//     PlcTask Inputs/GVL_Safety.SafetyInputs/bStageCollectRightDoorCh1 <-> Module 1 (FSOE)/FSoE Inputs/FSOE/FSIN Module 1.Input
//     PlcTask Inputs/GVL_Safety.SafetyInputs/bStageCollectRightDoorCh2 <-> Module 1 (FSOE)/FSoE Inputs/FSOE/FSIN Module 2.Input
//     PlcTask Inputs/GVL_Safety.SafetyInputs/bStageCollectRightDoorFdbk <-> Module 1 (FSOE)/FSoE Inputs/FSOE/FSIN Module 3.Input
//   TE1063/TE1063 Instance <-> Device 3 (EtherCAT)/Term 1 (EK1100)/Term 6 (EL1918)
//     PlcTask Inputs/GVL_IO.nEL1918T06State <-> InfoData/State
//     PlcTask Inputs/GVL_Safety.SafetyInputs/bD4AccessDoorIntlckOSSD1 <-> Module 1 (FSOE)/FSoE Inputs/FSOE/FSIN Module 3.Input
//     PlcTask Inputs/GVL_Safety.SafetyInputs/bD4AccessDoorIntlckOSSD2 <-> Module 1 (FSOE)/FSoE Inputs/FSOE/FSIN Module 4.Input
//     PlcTask Inputs/GVL_Safety.SafetyInputs/bD5AccessDoorIntlckOSSD1 <-> Module 1 (FSOE)/FSoE Inputs/FSOE/FSIN Module 5.Input
//     PlcTask Inputs/GVL_Safety.SafetyInputs/bD5AccessDoorIntlckOSSD2 <-> Module 1 (FSOE)/FSoE Inputs/FSOE/FSIN Module 6.Input
//     PlcTask Inputs/GVL_Safety.SafetyInputs/bD6AccessDoorIntlckOSSD1 <-> Module 1 (FSOE)/FSoE Inputs/FSOE/FSIN Module 7.Input
//     PlcTask Inputs/GVL_Safety.SafetyInputs/bD6AccessDoorIntlckOSSD2 <-> Module 1 (FSOE)/FSoE Inputs/FSOE/FSIN Module 8.Input
//     PlcTask Inputs/GVL_Safety.SafetyInputs/bFestoMS6DumpValveFdbk <-> Module 1 (FSOE)/FSoE Inputs/FSOE/FSIN Module 2.Input
//     PlcTask Inputs/GVL_Safety.SafetyInputs/bFestoMS6ValveFdbk <-> Module 1 (FSOE)/FSoE Inputs/FSOE/FSIN Module 1.Input
//   TE1063/TE1063 Instance <-> Device 3 (EtherCAT)/Term 1 (EK1100)/Term 7 (EL2904)
//     PlcTask Inputs/GVL_IO.nEL2904T07State <-> InfoData/State
//   TE1063/TE1063 Instance <-> Device 3 (EtherCAT)/Term 1 (EK1100)/Term 8 (EL2904)
//     PlcTask Inputs/GVL_IO.nEL2904T08State <-> InfoData/State
//   TE1063/TE1063 Instance <-> Device 3 (EtherCAT)/Term 1 (EK1100)/Term 9 (EL1809)
//     PlcTask Inputs/GVL_IO.gDigInputs/b24VPowerSupplyOK <-> Channel 3/Input
//     PlcTask Inputs/GVL_IO.gDigInputs/b48VPowerSupplyOK <-> Channel 5/Input
//     PlcTask Inputs/GVL_IO.gDigInputs/b24VPowerSupplyOKBck <-> Channel 4/Input
//     PlcTask Inputs/GVL_IO.gDigInputs/b48VPowerSupplyOKBck <-> Channel 12/Input
//     PlcTask Inputs/GVL_IO.gDigInputs/bCalibrationBoxPresent <-> Channel 13/Input
//     PlcTask Inputs/GVL_IO.gDigInputs/bSampleRecovery_Horizontal_Home <-> Channel 8/Input
//     PlcTask Inputs/GVL_IO.gDigInputs/bSampleRecovery_Vertical_Home <-> Channel 7/Input
//     PlcTask Inputs/GVL_IO.gDigInputs/bStageCollection_Home <-> Channel 6/Input
//     PlcTask Inputs/GVL_IO.gDigInputs/bStartButton <-> Channel 1/Input
//     PlcTask Inputs/GVL_IO.gDigInputs/bStopButton <-> Channel 2/Input
//     PlcTask Inputs/GVL_IO.gDigInputs/bThroatJigPresent <-> Channel 14/Input
//     PlcTask Inputs/GVL_IO.gDigInputs/bUPSReady <-> Channel 10/Input
//     PlcTask Inputs/GVL_IO.gDigInputs/bUPSReplaceBattery <-> Channel 11/Input
//     PlcTask Inputs/GVL_IO.gDigInputs/bWasteOverflowSensor <-> Channel 9/Input
//     PlcTask Inputs/GVL_IO.nEL1809T09State <-> InfoData/State
//   TE1063/TE1063 Instance <-> Device 3 (EtherCAT)/Term 22 (EK1100)
//     Task_Services Inputs/GVL_IO.nEK1100T22State <-> InfoData/State
//   TE1063/TE1063 Instance <-> Device 3 (EtherCAT)/Term 22 (EK1100)/Term 23 (EL7062)
//     PlcTask Inputs/GVL_Motion.aPumps[1].Linear.iHomeSensor <-> DRV Info data 3 Channel 1/Info data 3
//     PlcTask Inputs/GVL_Motion.aPumps[1].Linear.nState <-> InfoData/State
//     PlcTask Inputs/GVL_Motion.aPumps[1].Rotary.nState <-> InfoData/State
//   TE1063/TE1063 Instance <-> Device 3 (EtherCAT)/Term 22 (EK1100)/Term 24 (EL7062)
//     PlcTask Inputs/GVL_Motion.aPumps[2].Linear.iHomeSensor <-> DRV Info data 3 Channel 1/Info data 3
//     PlcTask Inputs/GVL_Motion.aPumps[2].Linear.nState <-> InfoData/State
//     PlcTask Inputs/GVL_Motion.aPumps[2].Rotary.nState <-> InfoData/State
//   TE1063/TE1063 Instance <-> Device 3 (EtherCAT)/Term 22 (EK1100)/Term 25 (EL7062)
//     PlcTask Inputs/GVL_Motion.aPumps[3].Linear.iHomeSensor <-> DRV Info data 3 Channel 1/Info data 3
//     PlcTask Inputs/GVL_Motion.aPumps[3].Linear.nState <-> InfoData/State
//     PlcTask Inputs/GVL_Motion.aPumps[3].Rotary.nState <-> InfoData/State
//   TE1063/TE1063 Instance <-> Device 3 (EtherCAT)/Term 22 (EK1100)/Term 26 (EL7062)
//     PlcTask Inputs/GVL_Motion.aPumps[4].Linear.iHomeSensor <-> DRV Info data 3 Channel 1/Info data 3
//     PlcTask Inputs/GVL_Motion.aPumps[4].Linear.nState <-> InfoData/State
//     PlcTask Inputs/GVL_Motion.aPumps[4].Rotary.nState <-> InfoData/State
//   TE1063/TE1063 Instance <-> Device 3 (EtherCAT)/Term 22 (EK1100)/Term 27 (EL7062)
//     PlcTask Inputs/GVL_Motion.aPumps[5].Linear.iHomeSensor <-> DRV Info data 3 Channel 1/Info data 3
//     PlcTask Inputs/GVL_Motion.aPumps[5].Linear.nState <-> InfoData/State
//     PlcTask Inputs/GVL_Motion.aPumps[5].Rotary.nState <-> InfoData/State
//   TE1063/TE1063 Instance <-> Device 3 (EtherCAT)/Term 22 (EK1100)/Term 28 (EL7062)
//     PlcTask Inputs/GVL_Motion.aPumps[6].Linear.iHomeSensor <-> DRV Info data 3 Channel 1/Info data 3
//     PlcTask Inputs/GVL_Motion.aPumps[6].Linear.nState <-> InfoData/State
//     PlcTask Inputs/GVL_Motion.aPumps[6].Rotary.nState <-> InfoData/State
//   TE1063/TE1063 Instance <-> Device 3 (EtherCAT)/Term 22 (EK1100)/Term 29 (EL7062)
//     PlcTask Inputs/GVL_Motion.aPumps[7].Linear.iHomeSensor <-> DRV Info data 3 Channel 1/Info data 3
//     PlcTask Inputs/GVL_Motion.aPumps[7].Linear.nState <-> InfoData/State
//     PlcTask Inputs/GVL_Motion.aPumps[7].Rotary.nState <-> InfoData/State
//   TE1063/TE1063 Instance <-> Device 3 (EtherCAT)/Term 22 (EK1100)/Term 30 (EL7062)
//     PlcTask Inputs/GVL_Motion.aPumps[8].Linear.iHomeSensor <-> DRV Info data 3 Channel 1/Info data 3
//     PlcTask Inputs/GVL_Motion.aPumps[8].Linear.nState <-> InfoData/State
//     PlcTask Inputs/GVL_Motion.aPumps[8].Rotary.nState <-> InfoData/State
//   TE1063/TE1063 Instance <-> Device 3 (EtherCAT)/Term 22 (EK1100)/Term 31 (EL7062)
//     PlcTask Inputs/GVL_Motion.aPumps[9].Linear.iHomeSensor <-> DRV Info data 3 Channel 1/Info data 3
//     PlcTask Inputs/GVL_Motion.aPumps[9].Linear.nState <-> InfoData/State
//     PlcTask Inputs/GVL_Motion.aPumps[9].Rotary.nState <-> InfoData/State
//   TE1063/TE1063 Instance <-> Device 3 (EtherCAT)/Term 22 (EK1100)/Term 32 (EL7062)
//     PlcTask Inputs/GVL_Motion.aPumps[10].Linear.iHomeSensor <-> DRV Info data 3 Channel 1/Info data 3
//     PlcTask Inputs/GVL_Motion.aPumps[10].Linear.nState <-> InfoData/State
//     PlcTask Inputs/GVL_Motion.aPumps[10].Rotary.nState <-> InfoData/State
//   TE1063/TE1063 Instance <-> Device 3 (EtherCAT)/Term 33 (AX8620-0000-0105)
//     Task_Services Inputs/GVL_IO.nAX8620T33State <-> InfoData/State
//   TE1063/TE1063 Instance <-> Device 3 (EtherCAT)/Term 33 (AX8620-0000-0105)/Drive 34 (AX8108-0100-0106)
//     PlcTask Inputs/GVL_Motion.M1Motor.nState <-> InfoData/State
//     PlcTask Outputs/GVL_Motion.M1Motor.bTS_ErrorAck <-> Device (Safety)/Standard Outputdata/ChA_Connection_Input.ERR_ACK FSoE Connection_3
//     PlcTask Outputs/GVL_Motion.M1Motor.bTS_Run <-> Device (Safety)/Standard Outputdata/ChA_Connection_Input.RUN FSoE Connection_2
//   TE1063/TE1063 Instance <-> Device 5 (EL6631)/dl-pn1
//     PlcTask Inputs/GVL_IO.gProfinetInput/bCurrentValueInvalid <-> API/Term 3 (GT2-***)/Subterm 5 (GT2-***)/Inputs/Sensor Status/Current_Value_Invalid
//     PlcTask Inputs/GVL_IO.gProfinetInput/bCurrentValueOverRange <-> API/Term 3 (GT2-***)/Subterm 5 (GT2-***)/Inputs/Sensor Status/Current_Value_Over_Range
//     PlcTask Inputs/GVL_IO.gProfinetInput/bCurrentValueUnerRange <-> API/Term 3 (GT2-***)/Subterm 5 (GT2-***)/Inputs/Sensor Status/Current_Value_Under_Range
//     PlcTask Inputs/GVL_IO.gProfinetInput/bErrorStatus <-> API/Term 3 (GT2-***)/Subterm 5 (GT2-***)/Inputs/Sensor Status/Error_Status
//     PlcTask Inputs/GVL_IO.gProfinetInput/bWarningStatus <-> API/Term 3 (GT2-***)/Subterm 5 (GT2-***)/Inputs/Sensor Status/Warning_Status
//     PlcTask Inputs/GVL_IO.gProfinetInput/iCurrentValue <-> API/Term 3 (GT2-***)/Subterm 5 (GT2-***)/Inputs/Current Value
//     PlcTask Inputs/GVL_IO.gProfinetInput/iPnIoBoxState <-> Inputs/PnIoBoxState
//   TE1063/TE1063 Instance <-> Device 6 (EtherCAT)/Box 10 (AMI8000-0100)
//     PlcTask Inputs/GVL_Motion.aValves[3].nState <-> InfoData/State
//     PlcTask Outputs/GVL_Safety.iM6STOErrorAck <-> Module 1 (SAFETY)/SAFETY Standard Outputdata/Standard In Var 3
//     PlcTask Outputs/GVL_Safety.iM6STORun <-> Module 1 (SAFETY)/SAFETY Standard Outputdata/Standard In Var 2
//   TE1063/TE1063 Instance <-> Device 6 (EtherCAT)/Box 11 (AMI8000-0100)
//     PlcTask Inputs/GVL_Motion.aValves[4].nState <-> InfoData/State
//     PlcTask Outputs/GVL_Safety.iM7STOErrorAck <-> Module 1 (SAFETY)/SAFETY Standard Outputdata/Standard In Var 3
//     PlcTask Outputs/GVL_Safety.iM7STORun <-> Module 1 (SAFETY)/SAFETY Standard Outputdata/Standard In Var 2
//   TE1063/TE1063 Instance <-> Device 6 (EtherCAT)/Box 12 (AMI8000-0100)
//     PlcTask Inputs/GVL_Motion.aValves[5].nState <-> InfoData/State
//     PlcTask Outputs/GVL_Safety.iM8STOErrorAck <-> Module 1 (SAFETY)/SAFETY Standard Outputdata/Standard In Var 3
//     PlcTask Outputs/GVL_Safety.iM8STORun <-> Module 1 (SAFETY)/SAFETY Standard Outputdata/Standard In Var 2
//   TE1063/TE1063 Instance <-> Device 6 (EtherCAT)/Box 8 (AMI8000-0100)
//     PlcTask Inputs/GVL_Motion.aValves[1].nState <-> InfoData/State
//     PlcTask Outputs/GVL_Safety.iM4STOErrorAck <-> Module 1 (SAFETY)/SAFETY Standard Outputdata/Standard In Var 3
//     PlcTask Outputs/GVL_Safety.iM4STORun <-> Module 1 (SAFETY)/SAFETY Standard Outputdata/Standard In Var 2
//   TE1063/TE1063 Instance <-> Device 6 (EtherCAT)/Box 9 (AMI8000-0100)
//     PlcTask Inputs/GVL_Motion.aValves[2].nState <-> InfoData/State
//     PlcTask Outputs/GVL_Safety.iM5STOErrorAck <-> Module 1 (SAFETY)/SAFETY Standard Outputdata/Standard In Var 3
//     PlcTask Outputs/GVL_Safety.iM5STORun <-> Module 1 (SAFETY)/SAFETY Standard Outputdata/Standard In Var 2
//   TE1063/TE1063 Instance <-> NC-Task 1 SAF/Axes/M1 Motor - SR Vertical
//     PlcTask Inputs/GVL_Motion.M1Motor.Axis.NcToPlc <-> Outputs/ToPlc
//     PlcTask Inputs/GVL_Motion.M1Motor.bMotionCommandsLocked <-> Outputs/ToPlc/StateDWord/MotionCommandsLocked
//     PlcTask Inputs/GVL_Motion.M1Motor.iError <-> Outputs/ToPlc/StateDWord/Error
//     PlcTask Inputs/GVL_Motion.M1Motor.iHomed <-> Outputs/ToPlc/StateDWord/Homed
//     PlcTask Inputs/GVL_Motion.M1Motor.iNotMoving <-> Outputs/ToPlc/StateDWord/NotMoving
//     PlcTask Inputs/GVL_Motion.M1Motor.iOperational <-> Outputs/ToPlc/StateDWord/Operational
//     PlcTask Inputs/GVL_Motion.M1Motor.nErrorCode <-> Outputs/ToPlc/ErrorCode
//     PlcTask Inputs/GVL_Motion.M1Motor.rActualPos <-> Outputs/ToPlc/ActPos
//     PlcTask Inputs/GVL_Motion.M1Motor.rActualTorque <-> Outputs/ToPlc/ActTorque
//     PlcTask Inputs/GVL_Motion.M1Motor.rActualVel <-> Outputs/ToPlc/ActVelo
//     PlcTask Outputs/GVL_Motion.M1Motor.Axis.PlcToNc <-> Inputs/FromPlc
//   TE1063/TE1063 Instance <-> NC-Task 1 SAF/Axes/M2 Motor - SC Vertical
//     PlcTask Inputs/GVL_Motion.M2Motor.Axis.NcToPlc <-> Outputs/ToPlc
//     PlcTask Inputs/GVL_Motion.M2Motor.bMotionCommandsLocked <-> Outputs/ToPlc/StateDWord/MotionCommandsLocked
//     PlcTask Inputs/GVL_Motion.M2Motor.iError <-> Outputs/ToPlc/StateDWord/Error
//     PlcTask Inputs/GVL_Motion.M2Motor.iHomed <-> Outputs/ToPlc/StateDWord/Homed
//     PlcTask Inputs/GVL_Motion.M2Motor.iNotMoving <-> Outputs/ToPlc/StateDWord/NotMoving
//     PlcTask Inputs/GVL_Motion.M2Motor.iOperational <-> Outputs/ToPlc/StateDWord/Operational
//     PlcTask Inputs/GVL_Motion.M2Motor.nErrorCode <-> Outputs/ToPlc/ErrorCode
//     PlcTask Inputs/GVL_Motion.M2Motor.rActualPos <-> Outputs/ToPlc/ActPos
//     PlcTask Inputs/GVL_Motion.M2Motor.rActualTorque <-> Outputs/ToPlc/ActTorque
//     PlcTask Inputs/GVL_Motion.M2Motor.rActualVel <-> Outputs/ToPlc/ActVelo
//     PlcTask Outputs/GVL_Motion.M2Motor.Axis.PlcToNc <-> Inputs/FromPlc
//   TE1063/TE1063 Instance <-> NC-Task 1 SAF/Axes/M3 Motor - SC Horizontal
//     PlcTask Inputs/GVL_Motion.M3Motor.Axis.NcToPlc <-> Outputs/ToPlc
//     PlcTask Inputs/GVL_Motion.M3Motor.bMotionCommandsLocked <-> Outputs/ToPlc/StateDWord/MotionCommandsLocked
//     PlcTask Inputs/GVL_Motion.M3Motor.iError <-> Outputs/ToPlc/StateDWord/Error
//     PlcTask Inputs/GVL_Motion.M3Motor.iHomed <-> Outputs/ToPlc/StateDWord/Homed
//     PlcTask Inputs/GVL_Motion.M3Motor.iNotMoving <-> Outputs/ToPlc/StateDWord/NotMoving
//     PlcTask Inputs/GVL_Motion.M3Motor.iOperational <-> Outputs/ToPlc/StateDWord/Operational
//     PlcTask Inputs/GVL_Motion.M3Motor.nErrorCode <-> Outputs/ToPlc/ErrorCode
//     PlcTask Inputs/GVL_Motion.M3Motor.rActualPos <-> Outputs/ToPlc/ActPos
//     PlcTask Inputs/GVL_Motion.M3Motor.rActualTorque <-> Outputs/ToPlc/ActTorque
//     PlcTask Inputs/GVL_Motion.M3Motor.rActualVel <-> Outputs/ToPlc/ActVelo
//     PlcTask Outputs/GVL_Motion.M3Motor.Axis.PlcToNc <-> Inputs/FromPlc
//   TE1063/TE1063 Instance <-> NC-Task 1 SAF/Axes/M4 Motor - Valve 1
//     PlcTask Inputs/GVL_Motion.aValves[1].Axis.NcToPlc <-> Outputs/ToPlc
//     PlcTask Inputs/GVL_Motion.aValves[1].bMotionCommandsLocked <-> Outputs/ToPlc/StateDWord/MotionCommandsLocked
//     PlcTask Inputs/GVL_Motion.aValves[1].iError <-> Outputs/ToPlc/StateDWord/Error
//     PlcTask Inputs/GVL_Motion.aValves[1].iHomed <-> Outputs/ToPlc/StateDWord/Homed
//     PlcTask Inputs/GVL_Motion.aValves[1].iNotMoving <-> Outputs/ToPlc/StateDWord/NotMoving
//     PlcTask Inputs/GVL_Motion.aValves[1].iOperational <-> Outputs/ToPlc/StateDWord/Operational
//     PlcTask Inputs/GVL_Motion.aValves[1].nErrorCode <-> Outputs/ToPlc/ErrorCode
//     PlcTask Inputs/GVL_Motion.aValves[1].rActualPos <-> Outputs/ToPlc/ActPos
//     PlcTask Inputs/GVL_Motion.aValves[1].rActualTorque <-> Outputs/ToPlc/ActTorque
//     PlcTask Inputs/GVL_Motion.aValves[1].rActualVel <-> Outputs/ToPlc/ActVelo
//     PlcTask Outputs/GVL_Motion.aValves[1].Axis.PlcToNc <-> Inputs/FromPlc
//   TE1063/TE1063 Instance <-> NC-Task 1 SAF/Axes/M5 Motor - Valve 2
//     PlcTask Inputs/GVL_Motion.aValves[2].Axis.NcToPlc <-> Outputs/ToPlc
//     PlcTask Inputs/GVL_Motion.aValves[2].bMotionCommandsLocked <-> Outputs/ToPlc/StateDWord/MotionCommandsLocked
//     PlcTask Inputs/GVL_Motion.aValves[2].iError <-> Outputs/ToPlc/StateDWord/Error
//     PlcTask Inputs/GVL_Motion.aValves[2].iHomed <-> Outputs/ToPlc/StateDWord/Homed
//     PlcTask Inputs/GVL_Motion.aValves[2].iNotMoving <-> Outputs/ToPlc/StateDWord/NotMoving
//     PlcTask Inputs/GVL_Motion.aValves[2].iOperational <-> Outputs/ToPlc/StateDWord/Operational
//     PlcTask Inputs/GVL_Motion.aValves[2].nErrorCode <-> Outputs/ToPlc/ErrorCode
//     PlcTask Inputs/GVL_Motion.aValves[2].rActualPos <-> Outputs/ToPlc/ActPos
//     PlcTask Inputs/GVL_Motion.aValves[2].rActualTorque <-> Outputs/ToPlc/ActTorque
//     PlcTask Inputs/GVL_Motion.aValves[2].rActualVel <-> Outputs/ToPlc/ActVelo
//     PlcTask Outputs/GVL_Motion.aValves[2].Axis.PlcToNc <-> Inputs/FromPlc
//   TE1063/TE1063 Instance <-> NC-Task 1 SAF/Axes/M6 Motor - Valve 3
//     PlcTask Inputs/GVL_Motion.aValves[3].Axis.NcToPlc <-> Outputs/ToPlc
//     PlcTask Inputs/GVL_Motion.aValves[3].bMotionCommandsLocked <-> Outputs/ToPlc/StateDWord/MotionCommandsLocked
//     PlcTask Inputs/GVL_Motion.aValves[3].iError <-> Outputs/ToPlc/StateDWord/Error
//     PlcTask Inputs/GVL_Motion.aValves[3].iHomed <-> Outputs/ToPlc/StateDWord/Homed
//     PlcTask Inputs/GVL_Motion.aValves[3].iNotMoving <-> Outputs/ToPlc/StateDWord/NotMoving
//     PlcTask Inputs/GVL_Motion.aValves[3].iOperational <-> Outputs/ToPlc/StateDWord/Operational
//     PlcTask Inputs/GVL_Motion.aValves[3].nErrorCode <-> Outputs/ToPlc/ErrorCode
//     PlcTask Inputs/GVL_Motion.aValves[3].rActualPos <-> Outputs/ToPlc/ActPos
//     PlcTask Inputs/GVL_Motion.aValves[3].rActualTorque <-> Outputs/ToPlc/ActTorque
//     PlcTask Inputs/GVL_Motion.aValves[3].rActualVel <-> Outputs/ToPlc/ActVelo
//     PlcTask Outputs/GVL_Motion.aValves[3].Axis.PlcToNc <-> Inputs/FromPlc
//   TE1063/TE1063 Instance <-> NC-Task 1 SAF/Axes/M7 Motor - Valve 4
//     PlcTask Inputs/GVL_Motion.aValves[4].Axis.NcToPlc <-> Outputs/ToPlc
//     PlcTask Inputs/GVL_Motion.aValves[4].bMotionCommandsLocked <-> Outputs/ToPlc/StateDWord/MotionCommandsLocked
//     PlcTask Inputs/GVL_Motion.aValves[4].iError <-> Outputs/ToPlc/StateDWord/Error
//     PlcTask Inputs/GVL_Motion.aValves[4].iHomed <-> Outputs/ToPlc/StateDWord/Homed
//     PlcTask Inputs/GVL_Motion.aValves[4].iNotMoving <-> Outputs/ToPlc/StateDWord/NotMoving
//     PlcTask Inputs/GVL_Motion.aValves[4].iOperational <-> Outputs/ToPlc/StateDWord/Operational
//     PlcTask Inputs/GVL_Motion.aValves[4].nErrorCode <-> Outputs/ToPlc/ErrorCode
//     PlcTask Inputs/GVL_Motion.aValves[4].rActualPos <-> Outputs/ToPlc/ActPos
//     PlcTask Inputs/GVL_Motion.aValves[4].rActualTorque <-> Outputs/ToPlc/ActTorque
//     PlcTask Inputs/GVL_Motion.aValves[4].rActualVel <-> Outputs/ToPlc/ActVelo
//     PlcTask Outputs/GVL_Motion.aValves[4].Axis.PlcToNc <-> Inputs/FromPlc
//   TE1063/TE1063 Instance <-> NC-Task 1 SAF/Axes/M8 Motor - Valve 5
//     PlcTask Inputs/GVL_Motion.aValves[5].Axis.NcToPlc <-> Outputs/ToPlc
//     PlcTask Inputs/GVL_Motion.aValves[5].bMotionCommandsLocked <-> Outputs/ToPlc/StateDWord/MotionCommandsLocked
//     PlcTask Inputs/GVL_Motion.aValves[5].iError <-> Outputs/ToPlc/StateDWord/Error
//     PlcTask Inputs/GVL_Motion.aValves[5].iHomed <-> Outputs/ToPlc/StateDWord/Homed
//     PlcTask Inputs/GVL_Motion.aValves[5].iNotMoving <-> Outputs/ToPlc/StateDWord/NotMoving
//     PlcTask Inputs/GVL_Motion.aValves[5].iOperational <-> Outputs/ToPlc/StateDWord/Operational
//     PlcTask Inputs/GVL_Motion.aValves[5].nErrorCode <-> Outputs/ToPlc/ErrorCode
//     PlcTask Inputs/GVL_Motion.aValves[5].rActualPos <-> Outputs/ToPlc/ActPos
//     PlcTask Inputs/GVL_Motion.aValves[5].rActualTorque <-> Outputs/ToPlc/ActTorque
//     PlcTask Inputs/GVL_Motion.aValves[5].rActualVel <-> Outputs/ToPlc/ActVelo
//     PlcTask Outputs/GVL_Motion.aValves[5].Axis.PlcToNc <-> Inputs/FromPlc
//   TE1063/TE1063 Instance <-> NC-Task 1 SAF/Axes/Pump 1 - Linear
//     PlcTask Inputs/GVL_Motion.aPumps[1].Linear.Axis.NcToPlc <-> Outputs/ToPlc
//     PlcTask Inputs/GVL_Motion.aPumps[1].Linear.iError <-> Outputs/ToPlc/StateDWord/Error
//     PlcTask Inputs/GVL_Motion.aPumps[1].Linear.iHomed <-> Outputs/ToPlc/StateDWord/Homed
//     PlcTask Inputs/GVL_Motion.aPumps[1].Linear.iNotMoving <-> Outputs/ToPlc/StateDWord/NotMoving
//     PlcTask Inputs/GVL_Motion.aPumps[1].Linear.iOperational <-> Outputs/ToPlc/StateDWord/Operational
//     PlcTask Inputs/GVL_Motion.aPumps[1].Linear.nErrorCode <-> Outputs/ToPlc/ErrorCode
//     PlcTask Inputs/GVL_Motion.aPumps[1].Linear.rActualPos <-> Outputs/ToPlc/ActPos
//     PlcTask Inputs/GVL_Motion.aPumps[1].Linear.rActualTorque <-> Outputs/ToPlc/ActTorque
//     PlcTask Inputs/GVL_Motion.aPumps[1].Linear.rActualVel <-> Outputs/ToPlc/ActVelo
//     PlcTask Outputs/GVL_Motion.aPumps[1].Linear.Axis.PlcToNc <-> Inputs/FromPlc
//   TE1063/TE1063 Instance <-> NC-Task 1 SAF/Axes/Pump 1 - Rotary
//     PlcTask Inputs/GVL_Motion.aPumps[1].Rotary.Axis.NcToPlc <-> Outputs/ToPlc
//     PlcTask Inputs/GVL_Motion.aPumps[1].Rotary.bMotionCommandsLocked <-> Outputs/ToPlc/StateDWord/MotionCommandsLocked
//     PlcTask Inputs/GVL_Motion.aPumps[1].Rotary.bNegativeDirection <-> Outputs/ToPlc/StateDWord/NegativeDirection
//     PlcTask Inputs/GVL_Motion.aPumps[1].Rotary.bPositiveDirection <-> Outputs/ToPlc/StateDWord/PositiveDirection
//     PlcTask Inputs/GVL_Motion.aPumps[1].Rotary.iError <-> Outputs/ToPlc/StateDWord/Error
//     PlcTask Inputs/GVL_Motion.aPumps[1].Rotary.iHomed <-> Outputs/ToPlc/StateDWord/Homed
//     PlcTask Inputs/GVL_Motion.aPumps[1].Rotary.iNotMoving <-> Outputs/ToPlc/StateDWord/NotMoving
//     PlcTask Inputs/GVL_Motion.aPumps[1].Rotary.iOperational <-> Outputs/ToPlc/StateDWord/Operational
//     PlcTask Inputs/GVL_Motion.aPumps[1].Rotary.nErrorCode <-> Outputs/ToPlc/ErrorCode
//     PlcTask Inputs/GVL_Motion.aPumps[1].Rotary.rActualPos <-> Outputs/ToPlc/ActPos
//     PlcTask Inputs/GVL_Motion.aPumps[1].Rotary.rActualTorque <-> Outputs/ToPlc/ActTorque
//     PlcTask Inputs/GVL_Motion.aPumps[1].Rotary.rActualVel <-> Outputs/ToPlc/ActVelo
//     PlcTask Outputs/GVL_Motion.aPumps[1].Rotary.Axis.PlcToNc <-> Inputs/FromPlc
//   TE1063/TE1063 Instance <-> NC-Task 1 SAF/Axes/Pump 10 - Linear
//     PlcTask Inputs/GVL_Motion.aPumps[10].Linear.Axis.NcToPlc <-> Outputs/ToPlc
//     PlcTask Inputs/GVL_Motion.aPumps[10].Linear.iError <-> Outputs/ToPlc/StateDWord/Error
//     PlcTask Inputs/GVL_Motion.aPumps[10].Linear.iHomed <-> Outputs/ToPlc/StateDWord/Homed
//     PlcTask Inputs/GVL_Motion.aPumps[10].Linear.iNotMoving <-> Outputs/ToPlc/StateDWord/NotMoving
//     PlcTask Inputs/GVL_Motion.aPumps[10].Linear.iOperational <-> Outputs/ToPlc/StateDWord/Operational
//     PlcTask Inputs/GVL_Motion.aPumps[10].Linear.nErrorCode <-> Outputs/ToPlc/ErrorCode
//     PlcTask Inputs/GVL_Motion.aPumps[10].Linear.rActualPos <-> Outputs/ToPlc/ActPos
//     PlcTask Inputs/GVL_Motion.aPumps[10].Linear.rActualTorque <-> Outputs/ToPlc/ActTorque
//     PlcTask Inputs/GVL_Motion.aPumps[10].Linear.rActualVel <-> Outputs/ToPlc/ActVelo
//     PlcTask Outputs/GVL_Motion.aPumps[10].Linear.Axis.PlcToNc <-> Inputs/FromPlc
//   TE1063/TE1063 Instance <-> NC-Task 1 SAF/Axes/Pump 10 - Rotary
//     PlcTask Inputs/GVL_Motion.aPumps[10].Rotary.Axis.NcToPlc <-> Outputs/ToPlc
//     PlcTask Inputs/GVL_Motion.aPumps[10].Rotary.bMotionCommandsLocked <-> Outputs/ToPlc/StateDWord/MotionCommandsLocked
//     PlcTask Inputs/GVL_Motion.aPumps[10].Rotary.bNegativeDirection <-> Outputs/ToPlc/StateDWord/NegativeDirection
//     PlcTask Inputs/GVL_Motion.aPumps[10].Rotary.bPositiveDirection <-> Outputs/ToPlc/StateDWord/PositiveDirection
//     PlcTask Inputs/GVL_Motion.aPumps[10].Rotary.iError <-> Outputs/ToPlc/StateDWord/Error
//     PlcTask Inputs/GVL_Motion.aPumps[10].Rotary.iHomed <-> Outputs/ToPlc/StateDWord/Homed
//     PlcTask Inputs/GVL_Motion.aPumps[10].Rotary.iNotMoving <-> Outputs/ToPlc/StateDWord/NotMoving
//     PlcTask Inputs/GVL_Motion.aPumps[10].Rotary.iOperational <-> Outputs/ToPlc/StateDWord/Operational
//     PlcTask Inputs/GVL_Motion.aPumps[10].Rotary.nErrorCode <-> Outputs/ToPlc/ErrorCode
//     PlcTask Inputs/GVL_Motion.aPumps[10].Rotary.rActualPos <-> Outputs/ToPlc/ActPos
//     PlcTask Inputs/GVL_Motion.aPumps[10].Rotary.rActualTorque <-> Outputs/ToPlc/ActTorque
//     PlcTask Inputs/GVL_Motion.aPumps[10].Rotary.rActualVel <-> Outputs/ToPlc/ActVelo
//     PlcTask Outputs/GVL_Motion.aPumps[10].Rotary.Axis.PlcToNc <-> Inputs/FromPlc
//   TE1063/TE1063 Instance <-> NC-Task 1 SAF/Axes/Pump 2 - Linear
//     PlcTask Inputs/GVL_Motion.aPumps[2].Linear.Axis.NcToPlc <-> Outputs/ToPlc
//     PlcTask Inputs/GVL_Motion.aPumps[2].Linear.iError <-> Outputs/ToPlc/StateDWord/Error
//     PlcTask Inputs/GVL_Motion.aPumps[2].Linear.iHomed <-> Outputs/ToPlc/StateDWord/Homed
//     PlcTask Inputs/GVL_Motion.aPumps[2].Linear.iNotMoving <-> Outputs/ToPlc/StateDWord/NotMoving
//     PlcTask Inputs/GVL_Motion.aPumps[2].Linear.iOperational <-> Outputs/ToPlc/StateDWord/Operational
//     PlcTask Inputs/GVL_Motion.aPumps[2].Linear.nErrorCode <-> Outputs/ToPlc/ErrorCode
//     PlcTask Inputs/GVL_Motion.aPumps[2].Linear.rActualPos <-> Outputs/ToPlc/ActPos
//     PlcTask Inputs/GVL_Motion.aPumps[2].Linear.rActualTorque <-> Outputs/ToPlc/ActTorque
//     PlcTask Inputs/GVL_Motion.aPumps[2].Linear.rActualVel <-> Outputs/ToPlc/ActVelo
//     PlcTask Outputs/GVL_Motion.aPumps[2].Linear.Axis.PlcToNc <-> Inputs/FromPlc
//   TE1063/TE1063 Instance <-> NC-Task 1 SAF/Axes/Pump 2 - Rotary
//     PlcTask Inputs/GVL_Motion.aPumps[2].Rotary.Axis.NcToPlc <-> Outputs/ToPlc
//     PlcTask Inputs/GVL_Motion.aPumps[2].Rotary.bMotionCommandsLocked <-> Outputs/ToPlc/StateDWord/MotionCommandsLocked
//     PlcTask Inputs/GVL_Motion.aPumps[2].Rotary.bNegativeDirection <-> Outputs/ToPlc/StateDWord/NegativeDirection
//     PlcTask Inputs/GVL_Motion.aPumps[2].Rotary.bPositiveDirection <-> Outputs/ToPlc/StateDWord/PositiveDirection
//     PlcTask Inputs/GVL_Motion.aPumps[2].Rotary.iError <-> Outputs/ToPlc/StateDWord/Error
//     PlcTask Inputs/GVL_Motion.aPumps[2].Rotary.iHomed <-> Outputs/ToPlc/StateDWord/Homed
//     PlcTask Inputs/GVL_Motion.aPumps[2].Rotary.iNotMoving <-> Outputs/ToPlc/StateDWord/NotMoving
//     PlcTask Inputs/GVL_Motion.aPumps[2].Rotary.iOperational <-> Outputs/ToPlc/StateDWord/Operational
//     PlcTask Inputs/GVL_Motion.aPumps[2].Rotary.nErrorCode <-> Outputs/ToPlc/ErrorCode
//     PlcTask Inputs/GVL_Motion.aPumps[2].Rotary.rActualPos <-> Outputs/ToPlc/ActPos
//     PlcTask Inputs/GVL_Motion.aPumps[2].Rotary.rActualTorque <-> Outputs/ToPlc/ActTorque
//     PlcTask Inputs/GVL_Motion.aPumps[2].Rotary.rActualVel <-> Outputs/ToPlc/ActVelo
//     PlcTask Outputs/GVL_Motion.aPumps[2].Rotary.Axis.PlcToNc <-> Inputs/FromPlc
//   TE1063/TE1063 Instance <-> NC-Task 1 SAF/Axes/Pump 3 - Linear
//     PlcTask Inputs/GVL_Motion.aPumps[3].Linear.Axis.NcToPlc <-> Outputs/ToPlc
//     PlcTask Inputs/GVL_Motion.aPumps[3].Linear.iError <-> Outputs/ToPlc/StateDWord/Error
//     PlcTask Inputs/GVL_Motion.aPumps[3].Linear.iHomed <-> Outputs/ToPlc/StateDWord/Homed
//     PlcTask Inputs/GVL_Motion.aPumps[3].Linear.iNotMoving <-> Outputs/ToPlc/StateDWord/NotMoving
//     PlcTask Inputs/GVL_Motion.aPumps[3].Linear.iOperational <-> Outputs/ToPlc/StateDWord/Operational
//     PlcTask Inputs/GVL_Motion.aPumps[3].Linear.nErrorCode <-> Outputs/ToPlc/ErrorCode
//     PlcTask Inputs/GVL_Motion.aPumps[3].Linear.rActualPos <-> Outputs/ToPlc/ActPos
//     PlcTask Inputs/GVL_Motion.aPumps[3].Linear.rActualTorque <-> Outputs/ToPlc/ActTorque
//     PlcTask Inputs/GVL_Motion.aPumps[3].Linear.rActualVel <-> Outputs/ToPlc/ActVelo
//     PlcTask Outputs/GVL_Motion.aPumps[3].Linear.Axis.PlcToNc <-> Inputs/FromPlc
//   TE1063/TE1063 Instance <-> NC-Task 1 SAF/Axes/Pump 3 - Rotary
//     PlcTask Inputs/GVL_Motion.aPumps[3].Rotary.Axis.NcToPlc <-> Outputs/ToPlc
//     PlcTask Inputs/GVL_Motion.aPumps[3].Rotary.bMotionCommandsLocked <-> Outputs/ToPlc/StateDWord/MotionCommandsLocked
//     PlcTask Inputs/GVL_Motion.aPumps[3].Rotary.bNegativeDirection <-> Outputs/ToPlc/StateDWord/NegativeDirection
//     PlcTask Inputs/GVL_Motion.aPumps[3].Rotary.bPositiveDirection <-> Outputs/ToPlc/StateDWord/PositiveDirection
//     PlcTask Inputs/GVL_Motion.aPumps[3].Rotary.iError <-> Outputs/ToPlc/StateDWord/Error
//     PlcTask Inputs/GVL_Motion.aPumps[3].Rotary.iHomed <-> Outputs/ToPlc/StateDWord/Homed
//     PlcTask Inputs/GVL_Motion.aPumps[3].Rotary.iNotMoving <-> Outputs/ToPlc/StateDWord/NotMoving
//     PlcTask Inputs/GVL_Motion.aPumps[3].Rotary.iOperational <-> Outputs/ToPlc/StateDWord/Operational
//     PlcTask Inputs/GVL_Motion.aPumps[3].Rotary.nErrorCode <-> Outputs/ToPlc/ErrorCode
//     PlcTask Inputs/GVL_Motion.aPumps[3].Rotary.rActualPos <-> Outputs/ToPlc/ActPos
//     PlcTask Inputs/GVL_Motion.aPumps[3].Rotary.rActualTorque <-> Outputs/ToPlc/ActTorque
//     PlcTask Inputs/GVL_Motion.aPumps[3].Rotary.rActualVel <-> Outputs/ToPlc/ActVelo
//     PlcTask Outputs/GVL_Motion.aPumps[3].Rotary.Axis.PlcToNc <-> Inputs/FromPlc
//   TE1063/TE1063 Instance <-> NC-Task 1 SAF/Axes/Pump 4 - Linear
//     PlcTask Inputs/GVL_Motion.aPumps[4].Linear.Axis.NcToPlc <-> Outputs/ToPlc
//     PlcTask Inputs/GVL_Motion.aPumps[4].Linear.iError <-> Outputs/ToPlc/StateDWord/Error
//     PlcTask Inputs/GVL_Motion.aPumps[4].Linear.iHomed <-> Outputs/ToPlc/StateDWord/Homed
//     PlcTask Inputs/GVL_Motion.aPumps[4].Linear.iNotMoving <-> Outputs/ToPlc/StateDWord/NotMoving
//     PlcTask Inputs/GVL_Motion.aPumps[4].Linear.iOperational <-> Outputs/ToPlc/StateDWord/Operational
//     PlcTask Inputs/GVL_Motion.aPumps[4].Linear.nErrorCode <-> Outputs/ToPlc/ErrorCode
//     PlcTask Inputs/GVL_Motion.aPumps[4].Linear.rActualPos <-> Outputs/ToPlc/ActPos
//     PlcTask Inputs/GVL_Motion.aPumps[4].Linear.rActualTorque <-> Outputs/ToPlc/ActTorque
//     PlcTask Inputs/GVL_Motion.aPumps[4].Linear.rActualVel <-> Outputs/ToPlc/ActVelo
//     PlcTask Outputs/GVL_Motion.aPumps[4].Linear.Axis.PlcToNc <-> Inputs/FromPlc
//   TE1063/TE1063 Instance <-> NC-Task 1 SAF/Axes/Pump 4 - Rotary
//     PlcTask Inputs/GVL_Motion.aPumps[4].Rotary.Axis.NcToPlc <-> Outputs/ToPlc
//     PlcTask Inputs/GVL_Motion.aPumps[4].Rotary.bMotionCommandsLocked <-> Outputs/ToPlc/StateDWord/MotionCommandsLocked
//     PlcTask Inputs/GVL_Motion.aPumps[4].Rotary.bNegativeDirection <-> Outputs/ToPlc/StateDWord/NegativeDirection
//     PlcTask Inputs/GVL_Motion.aPumps[4].Rotary.bPositiveDirection <-> Outputs/ToPlc/StateDWord/PositiveDirection
//     PlcTask Inputs/GVL_Motion.aPumps[4].Rotary.iError <-> Outputs/ToPlc/StateDWord/Error
//     PlcTask Inputs/GVL_Motion.aPumps[4].Rotary.iHomed <-> Outputs/ToPlc/StateDWord/Homed
//     PlcTask Inputs/GVL_Motion.aPumps[4].Rotary.iNotMoving <-> Outputs/ToPlc/StateDWord/NotMoving
//     PlcTask Inputs/GVL_Motion.aPumps[4].Rotary.iOperational <-> Outputs/ToPlc/StateDWord/Operational
//     PlcTask Inputs/GVL_Motion.aPumps[4].Rotary.nErrorCode <-> Outputs/ToPlc/ErrorCode
//     PlcTask Inputs/GVL_Motion.aPumps[4].Rotary.rActualPos <-> Outputs/ToPlc/ActPos
//     PlcTask Inputs/GVL_Motion.aPumps[4].Rotary.rActualTorque <-> Outputs/ToPlc/ActTorque
//     PlcTask Inputs/GVL_Motion.aPumps[4].Rotary.rActualVel <-> Outputs/ToPlc/ActVelo
//     PlcTask Outputs/GVL_Motion.aPumps[4].Rotary.Axis.PlcToNc <-> Inputs/FromPlc
//   TE1063/TE1063 Instance <-> NC-Task 1 SAF/Axes/Pump 5 - Linear
//     PlcTask Inputs/GVL_Motion.aPumps[5].Linear.Axis.NcToPlc <-> Outputs/ToPlc
//     PlcTask Inputs/GVL_Motion.aPumps[5].Linear.iError <-> Outputs/ToPlc/StateDWord/Error
//     PlcTask Inputs/GVL_Motion.aPumps[5].Linear.iHomed <-> Outputs/ToPlc/StateDWord/Homed
//     PlcTask Inputs/GVL_Motion.aPumps[5].Linear.iNotMoving <-> Outputs/ToPlc/StateDWord/NotMoving
//     PlcTask Inputs/GVL_Motion.aPumps[5].Linear.iOperational <-> Outputs/ToPlc/StateDWord/Operational
//     PlcTask Inputs/GVL_Motion.aPumps[5].Linear.nErrorCode <-> Outputs/ToPlc/ErrorCode
//     PlcTask Inputs/GVL_Motion.aPumps[5].Linear.rActualPos <-> Outputs/ToPlc/ActPos
//     PlcTask Inputs/GVL_Motion.aPumps[5].Linear.rActualTorque <-> Outputs/ToPlc/ActTorque
//     PlcTask Inputs/GVL_Motion.aPumps[5].Linear.rActualVel <-> Outputs/ToPlc/ActVelo
//     PlcTask Outputs/GVL_Motion.aPumps[5].Linear.Axis.PlcToNc <-> Inputs/FromPlc
//   TE1063/TE1063 Instance <-> NC-Task 1 SAF/Axes/Pump 5 - Rotary
//     PlcTask Inputs/GVL_Motion.aPumps[5].Rotary.Axis.NcToPlc <-> Outputs/ToPlc
//     PlcTask Inputs/GVL_Motion.aPumps[5].Rotary.bMotionCommandsLocked <-> Outputs/ToPlc/StateDWord/MotionCommandsLocked
//     PlcTask Inputs/GVL_Motion.aPumps[5].Rotary.bNegativeDirection <-> Outputs/ToPlc/StateDWord/NegativeDirection
//     PlcTask Inputs/GVL_Motion.aPumps[5].Rotary.bPositiveDirection <-> Outputs/ToPlc/StateDWord/PositiveDirection
//     PlcTask Inputs/GVL_Motion.aPumps[5].Rotary.iError <-> Outputs/ToPlc/StateDWord/Error
//     PlcTask Inputs/GVL_Motion.aPumps[5].Rotary.iHomed <-> Outputs/ToPlc/StateDWord/Homed
//     PlcTask Inputs/GVL_Motion.aPumps[5].Rotary.iNotMoving <-> Outputs/ToPlc/StateDWord/NotMoving
//     PlcTask Inputs/GVL_Motion.aPumps[5].Rotary.iOperational <-> Outputs/ToPlc/StateDWord/Operational
//     PlcTask Inputs/GVL_Motion.aPumps[5].Rotary.nErrorCode <-> Outputs/ToPlc/ErrorCode
//     PlcTask Inputs/GVL_Motion.aPumps[5].Rotary.rActualPos <-> Outputs/ToPlc/ActPos
//     PlcTask Inputs/GVL_Motion.aPumps[5].Rotary.rActualTorque <-> Outputs/ToPlc/ActTorque
//     PlcTask Inputs/GVL_Motion.aPumps[5].Rotary.rActualVel <-> Outputs/ToPlc/ActVelo
//     PlcTask Outputs/GVL_Motion.aPumps[5].Rotary.Axis.PlcToNc <-> Inputs/FromPlc
//   TE1063/TE1063 Instance <-> NC-Task 1 SAF/Axes/Pump 6 - Linear
//     PlcTask Inputs/GVL_Motion.aPumps[6].Linear.Axis.NcToPlc <-> Outputs/ToPlc
//     PlcTask Inputs/GVL_Motion.aPumps[6].Linear.iError <-> Outputs/ToPlc/StateDWord/Error
//     PlcTask Inputs/GVL_Motion.aPumps[6].Linear.iHomed <-> Outputs/ToPlc/StateDWord/Homed
//     PlcTask Inputs/GVL_Motion.aPumps[6].Linear.iNotMoving <-> Outputs/ToPlc/StateDWord/NotMoving
//     PlcTask Inputs/GVL_Motion.aPumps[6].Linear.iOperational <-> Outputs/ToPlc/StateDWord/Operational
//     PlcTask Inputs/GVL_Motion.aPumps[6].Linear.nErrorCode <-> Outputs/ToPlc/ErrorCode
//     PlcTask Inputs/GVL_Motion.aPumps[6].Linear.rActualPos <-> Outputs/ToPlc/ActPos
//     PlcTask Inputs/GVL_Motion.aPumps[6].Linear.rActualTorque <-> Outputs/ToPlc/ActTorque
//     PlcTask Inputs/GVL_Motion.aPumps[6].Linear.rActualVel <-> Outputs/ToPlc/ActVelo
//     PlcTask Outputs/GVL_Motion.aPumps[6].Linear.Axis.PlcToNc <-> Inputs/FromPlc
//   TE1063/TE1063 Instance <-> NC-Task 1 SAF/Axes/Pump 6 - Rotary
//     PlcTask Inputs/GVL_Motion.aPumps[6].Rotary.Axis.NcToPlc <-> Outputs/ToPlc
//     PlcTask Inputs/GVL_Motion.aPumps[6].Rotary.bMotionCommandsLocked <-> Outputs/ToPlc/StateDWord/MotionCommandsLocked
//     PlcTask Inputs/GVL_Motion.aPumps[6].Rotary.bNegativeDirection <-> Outputs/ToPlc/StateDWord/NegativeDirection
//     PlcTask Inputs/GVL_Motion.aPumps[6].Rotary.bPositiveDirection <-> Outputs/ToPlc/StateDWord/PositiveDirection
//     PlcTask Inputs/GVL_Motion.aPumps[6].Rotary.iError <-> Outputs/ToPlc/StateDWord/Error
//     PlcTask Inputs/GVL_Motion.aPumps[6].Rotary.iHomed <-> Outputs/ToPlc/StateDWord/Homed
//     PlcTask Inputs/GVL_Motion.aPumps[6].Rotary.iNotMoving <-> Outputs/ToPlc/StateDWord/NotMoving
//     PlcTask Inputs/GVL_Motion.aPumps[6].Rotary.iOperational <-> Outputs/ToPlc/StateDWord/Operational
//     PlcTask Inputs/GVL_Motion.aPumps[6].Rotary.nErrorCode <-> Outputs/ToPlc/ErrorCode
//     PlcTask Inputs/GVL_Motion.aPumps[6].Rotary.rActualPos <-> Outputs/ToPlc/ActPos
//     PlcTask Inputs/GVL_Motion.aPumps[6].Rotary.rActualTorque <-> Outputs/ToPlc/ActTorque
//     PlcTask Inputs/GVL_Motion.aPumps[6].Rotary.rActualVel <-> Outputs/ToPlc/ActVelo
//     PlcTask Outputs/GVL_Motion.aPumps[6].Rotary.Axis.PlcToNc <-> Inputs/FromPlc
//   TE1063/TE1063 Instance <-> NC-Task 1 SAF/Axes/Pump 7 - Linear
//     PlcTask Inputs/GVL_Motion.aPumps[7].Linear.Axis.NcToPlc <-> Outputs/ToPlc
//     PlcTask Inputs/GVL_Motion.aPumps[7].Linear.iError <-> Outputs/ToPlc/StateDWord/Error
//     PlcTask Inputs/GVL_Motion.aPumps[7].Linear.iHomed <-> Outputs/ToPlc/StateDWord/Homed
//     PlcTask Inputs/GVL_Motion.aPumps[7].Linear.iNotMoving <-> Outputs/ToPlc/StateDWord/NotMoving
//     PlcTask Inputs/GVL_Motion.aPumps[7].Linear.iOperational <-> Outputs/ToPlc/StateDWord/Operational
//     PlcTask Inputs/GVL_Motion.aPumps[7].Linear.nErrorCode <-> Outputs/ToPlc/ErrorCode
//     PlcTask Inputs/GVL_Motion.aPumps[7].Linear.rActualPos <-> Outputs/ToPlc/ActPos
//     PlcTask Inputs/GVL_Motion.aPumps[7].Linear.rActualTorque <-> Outputs/ToPlc/ActTorque
//     PlcTask Inputs/GVL_Motion.aPumps[7].Linear.rActualVel <-> Outputs/ToPlc/ActVelo
//     PlcTask Outputs/GVL_Motion.aPumps[7].Linear.Axis.PlcToNc <-> Inputs/FromPlc
//   TE1063/TE1063 Instance <-> NC-Task 1 SAF/Axes/Pump 7 - Rotary
//     PlcTask Inputs/GVL_Motion.aPumps[7].Rotary.Axis.NcToPlc <-> Outputs/ToPlc
//     PlcTask Inputs/GVL_Motion.aPumps[7].Rotary.bMotionCommandsLocked <-> Outputs/ToPlc/StateDWord/MotionCommandsLocked
//     PlcTask Inputs/GVL_Motion.aPumps[7].Rotary.bNegativeDirection <-> Outputs/ToPlc/StateDWord/NegativeDirection
//     PlcTask Inputs/GVL_Motion.aPumps[7].Rotary.bPositiveDirection <-> Outputs/ToPlc/StateDWord/PositiveDirection
//     PlcTask Inputs/GVL_Motion.aPumps[7].Rotary.iError <-> Outputs/ToPlc/StateDWord/Error
//     PlcTask Inputs/GVL_Motion.aPumps[7].Rotary.iHomed <-> Outputs/ToPlc/StateDWord/Homed
//     PlcTask Inputs/GVL_Motion.aPumps[7].Rotary.iNotMoving <-> Outputs/ToPlc/StateDWord/NotMoving
//     PlcTask Inputs/GVL_Motion.aPumps[7].Rotary.iOperational <-> Outputs/ToPlc/StateDWord/Operational
//     PlcTask Inputs/GVL_Motion.aPumps[7].Rotary.nErrorCode <-> Outputs/ToPlc/ErrorCode
//     PlcTask Inputs/GVL_Motion.aPumps[7].Rotary.rActualPos <-> Outputs/ToPlc/ActPos
//     PlcTask Inputs/GVL_Motion.aPumps[7].Rotary.rActualTorque <-> Outputs/ToPlc/ActTorque
//     PlcTask Inputs/GVL_Motion.aPumps[7].Rotary.rActualVel <-> Outputs/ToPlc/ActVelo
//     PlcTask Outputs/GVL_Motion.aPumps[7].Rotary.Axis.PlcToNc <-> Inputs/FromPlc
//   TE1063/TE1063 Instance <-> NC-Task 1 SAF/Axes/Pump 8 - Linear
//     PlcTask Inputs/GVL_Motion.aPumps[8].Linear.Axis.NcToPlc <-> Outputs/ToPlc
//     PlcTask Inputs/GVL_Motion.aPumps[8].Linear.iError <-> Outputs/ToPlc/StateDWord/Error
//     PlcTask Inputs/GVL_Motion.aPumps[8].Linear.iHomed <-> Outputs/ToPlc/StateDWord/Homed
//     PlcTask Inputs/GVL_Motion.aPumps[8].Linear.iNotMoving <-> Outputs/ToPlc/StateDWord/NotMoving
//     PlcTask Inputs/GVL_Motion.aPumps[8].Linear.iOperational <-> Outputs/ToPlc/StateDWord/Operational
//     PlcTask Inputs/GVL_Motion.aPumps[8].Linear.nErrorCode <-> Outputs/ToPlc/ErrorCode
//     PlcTask Inputs/GVL_Motion.aPumps[8].Linear.rActualPos <-> Outputs/ToPlc/ActPos
//     PlcTask Inputs/GVL_Motion.aPumps[8].Linear.rActualTorque <-> Outputs/ToPlc/ActTorque
//     PlcTask Inputs/GVL_Motion.aPumps[8].Linear.rActualVel <-> Outputs/ToPlc/ActVelo
//     PlcTask Outputs/GVL_Motion.aPumps[8].Linear.Axis.PlcToNc <-> Inputs/FromPlc
//   TE1063/TE1063 Instance <-> NC-Task 1 SAF/Axes/Pump 8 - Rotary
//     PlcTask Inputs/GVL_Motion.aPumps[8].Rotary.Axis.NcToPlc <-> Outputs/ToPlc
//     PlcTask Inputs/GVL_Motion.aPumps[8].Rotary.bMotionCommandsLocked <-> Outputs/ToPlc/StateDWord/MotionCommandsLocked
//     PlcTask Inputs/GVL_Motion.aPumps[8].Rotary.bNegativeDirection <-> Outputs/ToPlc/StateDWord/NegativeDirection
//     PlcTask Inputs/GVL_Motion.aPumps[8].Rotary.bPositiveDirection <-> Outputs/ToPlc/StateDWord/PositiveDirection
//     PlcTask Inputs/GVL_Motion.aPumps[8].Rotary.iError <-> Outputs/ToPlc/StateDWord/Error
//     PlcTask Inputs/GVL_Motion.aPumps[8].Rotary.iHomed <-> Outputs/ToPlc/StateDWord/Homed
//     PlcTask Inputs/GVL_Motion.aPumps[8].Rotary.iNotMoving <-> Outputs/ToPlc/StateDWord/NotMoving
//     PlcTask Inputs/GVL_Motion.aPumps[8].Rotary.iOperational <-> Outputs/ToPlc/StateDWord/Operational
//     PlcTask Inputs/GVL_Motion.aPumps[8].Rotary.nErrorCode <-> Outputs/ToPlc/ErrorCode
//     PlcTask Inputs/GVL_Motion.aPumps[8].Rotary.rActualPos <-> Outputs/ToPlc/ActPos
//     PlcTask Inputs/GVL_Motion.aPumps[8].Rotary.rActualTorque <-> Outputs/ToPlc/ActTorque
//     PlcTask Inputs/GVL_Motion.aPumps[8].Rotary.rActualVel <-> Outputs/ToPlc/ActVelo
//     PlcTask Outputs/GVL_Motion.aPumps[8].Rotary.Axis.PlcToNc <-> Inputs/FromPlc
//   TE1063/TE1063 Instance <-> NC-Task 1 SAF/Axes/Pump 9 - Linear
//     PlcTask Inputs/GVL_Motion.aPumps[9].Linear.Axis.NcToPlc <-> Outputs/ToPlc
//     PlcTask Inputs/GVL_Motion.aPumps[9].Linear.iError <-> Outputs/ToPlc/StateDWord/Error
//     PlcTask Inputs/GVL_Motion.aPumps[9].Linear.iHomed <-> Outputs/ToPlc/StateDWord/Homed
//     PlcTask Inputs/GVL_Motion.aPumps[9].Linear.iNotMoving <-> Outputs/ToPlc/StateDWord/NotMoving
//     PlcTask Inputs/GVL_Motion.aPumps[9].Linear.iOperational <-> Outputs/ToPlc/StateDWord/Operational
//     PlcTask Inputs/GVL_Motion.aPumps[9].Linear.nErrorCode <-> Outputs/ToPlc/ErrorCode
//     PlcTask Inputs/GVL_Motion.aPumps[9].Linear.rActualPos <-> Outputs/ToPlc/ActPos
//     PlcTask Inputs/GVL_Motion.aPumps[9].Linear.rActualTorque <-> Outputs/ToPlc/ActTorque
//     PlcTask Inputs/GVL_Motion.aPumps[9].Linear.rActualVel <-> Outputs/ToPlc/ActVelo
//     PlcTask Outputs/GVL_Motion.aPumps[9].Linear.Axis.PlcToNc <-> Inputs/FromPlc
//   TE1063/TE1063 Instance <-> NC-Task 1 SAF/Axes/Pump 9 - Rotary
//     PlcTask Inputs/GVL_Motion.aPumps[9].Rotary.Axis.NcToPlc <-> Outputs/ToPlc
//     PlcTask Inputs/GVL_Motion.aPumps[9].Rotary.bMotionCommandsLocked <-> Outputs/ToPlc/StateDWord/MotionCommandsLocked
//     PlcTask Inputs/GVL_Motion.aPumps[9].Rotary.bNegativeDirection <-> Outputs/ToPlc/StateDWord/NegativeDirection
//     PlcTask Inputs/GVL_Motion.aPumps[9].Rotary.bPositiveDirection <-> Outputs/ToPlc/StateDWord/PositiveDirection
//     PlcTask Inputs/GVL_Motion.aPumps[9].Rotary.iError <-> Outputs/ToPlc/StateDWord/Error
//     PlcTask Inputs/GVL_Motion.aPumps[9].Rotary.iHomed <-> Outputs/ToPlc/StateDWord/Homed
//     PlcTask Inputs/GVL_Motion.aPumps[9].Rotary.iNotMoving <-> Outputs/ToPlc/StateDWord/NotMoving
//     PlcTask Inputs/GVL_Motion.aPumps[9].Rotary.iOperational <-> Outputs/ToPlc/StateDWord/Operational
//     PlcTask Inputs/GVL_Motion.aPumps[9].Rotary.nErrorCode <-> Outputs/ToPlc/ErrorCode
//     PlcTask Inputs/GVL_Motion.aPumps[9].Rotary.rActualPos <-> Outputs/ToPlc/ActPos
//     PlcTask Inputs/GVL_Motion.aPumps[9].Rotary.rActualTorque <-> Outputs/ToPlc/ActTorque
//     PlcTask Inputs/GVL_Motion.aPumps[9].Rotary.rActualVel <-> Outputs/ToPlc/ActVelo
//     PlcTask Outputs/GVL_Motion.aPumps[9].Rotary.Axis.PlcToNc <-> Inputs/FromPlc

CONFIGURATION TE1063
    RESOURCE PLC ON TwinCAT3
        TASK PlcTask(INTERVAL := T#10ms, PRIORITY := 10);
        TASK Task_Events(INTERVAL := T#250ms, PRIORITY := 14);
        TASK Task_HMI(INTERVAL := T#100000us, PRIORITY := 12);
        TASK Task_Services(INTERVAL := T#1000ms, PRIORITY := 16);
        PROGRAM MAIN_Control WITH PlcTask : MAIN_Control;
        PROGRAM MAIN_Events WITH Task_Events : MAIN_Events;
        PROGRAM MAIN_HMI WITH Task_HMI : MAIN_HMI;
        PROGRAM MAIN_Services WITH Task_Services : MAIN_Services;
    END_RESOURCE
END_CONFIGURATION

// ---- DUTs/AlarmEventLogger/E_Events.TcDUT
{attribute 'qualified_only'}
{attribute 'strict'}
TYPE E_Events :
(
	// Enum for events and alarms different severity
	INFO 	:= 1,
	WARNING := 2,
	ERROR	:= 3,
	CRITICAL:= 4
);
END_TYPE

// ---- DUTs/AlarmEventLogger/ST_GeneralAlarm.TcDUT
TYPE ST_GeneralAlarm :
STRUCT
	bEmergencyStopActive : BOOL := FALSE; // Alarm status active
	bSystemFault         : BOOL := FALSE; // General system failure
	sMessage             : STRING(80) := ''; // General alarm message
END_STRUCT
END_TYPE

// ---- DUTs/AlarmEventLogger/ST_ValveError.TcDUT
TYPE ST_ValveError :
STRUCT
	bActive       : BOOL := FALSE; // Indicates active error in the valves
	nValveIndex   : INT  := 0;     // Valve index with error (1 to 5)
	nErrorID      : UDINT := 0;    // Error code returned
	sErrorMessage : STRING(80) := '';
END_STRUCT
END_TYPE

// ---- DUTs/AutoCycle/E_MachineStates.TcDUT
{attribute 'qualified_only'}
{attribute 'strict'}
TYPE E_MachineStates :
(
	INIT 			:= 100,         // Initialization 
    CHECK_AIR_FLOW 	:= 110,         // Air Flow Verifying 
    SEAL_STAGES 	:= 130,         // Seal Stages/plates cycle 
    LEAK_TEST 		:= 140,         // Leak Test cycle 
	PRIME_SOLVENT	:= 150,			// Prime Solvents cycle 
    RECOVERY_PHASE 	:= 160,         // Recovery Cycle 
    WASHING_PHASE 	:= 170,         // Washing Cycle
    DRYING_PHASE 	:= 180,         // Drying Cycle
    POST_EXECUTION 	:= 190,         // Post Execution
	PAUSE_STATE		:= 200,			// Pause/Hold State
    ERROR_STATE 	:= 99           // Error State 
);
END_TYPE

// ---- DUTs/AutoCycle/E_PrimeSolventState.TcDUT
{attribute 'qualified_only'}
{attribute 'strict'}
TYPE E_PrimeSolventState :
(
	PS_Idle := 0,
    PS_Solvent1 := 10,
    PS_Solvent2 := 20,
    PS_Solvent3 := 30,
    PS_Solvent4 := 40,
    PS_Completed := 100
);
END_TYPE

// ---- DUTs/AutoCycle/E_RecoveryState.TcDUT
{attribute 'qualified_only'}
{attribute 'strict'}
TYPE E_RecoveryState :
(

	Idle 						:= 0,
	Metering_Solvent1 			:= 1,
	Recirculate_Solvent1 		:= 2,
	Solvent_Soak 				:= 3,
	Cleaning_Lines_S1 			:= 4,
	Metering_Solvent2 			:= 5,
	AgitateTime1				:= 6,
	Mix_Solvent1_2 				:= 7,
	Cleaning_Lines_S1_S2 		:= 8,
	AgitateTime2				:= 9,
	Prime_Needles 				:= 10,
	Fill_Vials_Row_1 			:= 11,
	Fill_Vials_Row_2 			:= 12,
	Fill_Vials_Row_3 			:= 13,
	Fill_Vials_Row_4 			:= 14,
	Waste_Remaining_Solvent 	:= 15,
	Completed 					:= 16,
	Error						:= 17

);
END_TYPE

// ---- DUTs/AutoCycle/E_WashingState.TcDUT
{attribute 'qualified_only'}
{attribute 'strict'}
TYPE E_WashingState :
(
	Idle 				:= 0,
	Metering_Wash1		:= 1,
	Recirculate_Wash1	:= 2,
	Cleaning_Lines_W1	:= 3,
	Waste_Wash1			:= 4,
	Metering_Wash2		:= 5,
	Recirculate_Wash2	:= 6,
	Cleaning_Lines_W2	:= 7,
	Waste_Wash2			:= 8,
	Completed 			:= 9,
	Error				:= 10
	
);
END_TYPE

// ---- DUTs/Calibration/E_LeakTestState.TcDUT
{attribute 'qualified_only'}
{attribute 'strict'}
TYPE E_LeakTestState :
(
	IDLE := 0,
	PRESSURE_UP := 1,
	HOLD_PRESSURE :=2
);
END_TYPE

// ---- DUTs/Calibration/E_PState.TcDUT
{attribute 'qualified_only'}
{attribute 'strict'}
TYPE E_PState :
(
	Init, 
	SealIssue, 
	SealWait, 
	OpenValves, 
	Done, 
	Fault
);
END_TYPE

// ---- DUTs/Calibration/E_StopState.TcDUT
{attribute 'qualified_only'}
{attribute 'strict'}
TYPE E_StopState :
(
	Init, 
	StopMotor, 
	CloseSolenoids, 
	Delay, 
	ResetMotor, 
	MoveHome, 
	Done
);
END_TYPE

// ---- DUTs/Calibration/E_CalibrationStatus.TcDUT
{attribute 'qualified_only'}
{attribute 'strict'}
TYPE E_CalibrationStatus :
(
	IDLE,
    PENDING,
    RUNNING,
    PASSED,
    FAILED,
    ADJUSTMENT_NEEDED,
	UNKNOWN
);
END_TYPE

// ---- DUTs/Calibration/E_CalibStep.TcDUT
{attribute 'qualified_only'}
{attribute 'strict'}
TYPE E_CalibStep :
(
	IDLE 				:= 0, 	// Idle State
    DELAY 				:= 5, 	// Delay state depending on delay time to start calibration on HMI
	CHECKING_WEIGH 		:= 10,	// Checking if the calibration box is on the correct weight
	POSITION_MOTORS 	:= 20,	// Position the motors M2 and M3 to calibration position
	POSITION_VALVES 	:= 30,	// Position Valves into calibration position
	FILLJAR_FORWARD 	:= 40,	// Fill the jars first with the volume in the HMI plus tubing dead volume
	WEIGH_BEFORE 		:= 50,	// Request calibration box weight [Tare weight]
	WITHDRAW_BACKWARDS 	:= 60,	// Pump back to calibration box the amount of liquid into the HMI
	WEIGH_AFTER 		:= 70,	// Request the calibration box weight after pumping [Gross Weight]  
	RETURN_FORWARD 		:= 80,	// Return to the jar the same amount of liquid that was dosed by the pump
	PUMPFACTOR_ADJUST	:= 85,	// Adjust the pump factor if the net volume is less than 10% off the target 
	PUMPFACTOR_FAILED	:= 86,	// If pump factor number of adjustments is greater than allowable failures
	FEED_HMI_RESULTS	:= 90,  // Feed HMI controls with pump results 
	EMPTYJAR_BACKWARDS 	:= 95,	// Empty the Jar with 60% more revs to make sure everything was cleaned
	NEXT_PUMP 			:= 100,	// Going to next pump calibration
	HOMING_MOTORS 		:= 110,	// Moving the motors M2 and M3 back to home position
	REPORT_INFO_UPDATE	:= 120, // Step where all the reports info are updated
	AIR_DRY_TIME		:= 130, // Air Dry Time when calibration is finished
	CALBOX_ATTENTION	:= 170, // Step where the FB waits for someone fill up the calibration box
	SCALE_ATTENTION		:= 180, // Step where the FB waits for human interaction in the scale
	COMPLETE 			:= 200,	// Complete state
	ERROR 				:= 300	// Error state
);
END_TYPE

// ---- DUTs/Calibration/E_ScaleCmd.TcDUT
{attribute 'qualified_only'}
{attribute 'strict'}
TYPE E_ScaleCmd :
(
	ScaleCmd_None, 
	ScaleCmd_SI, 
	ScaleCmd_S, 
	ScaleCmd_T, 
	ScaleCmd_TA, 
	ScaleCmd_TAC
);
END_TYPE

// ---- DUTs/Calibration/E_SolventType.TcDUT
{attribute 'qualified_only'}
{attribute 'strict'}
TYPE E_SolventType :
(
	Solvent1,
	Solvent2,
	Solvent3,
	Solvent4,
	Solvent5
);
END_TYPE

// ---- DUTs/Calibration/ST_CalibrationData.TcDUT
TYPE ST_CalibrationData :
STRUCT
	dDateTime 		: STRING(32);
	iPumpNumber 	: USINT;
	sStep			: STRING(64);
	rTareWeigth		: LREAL;
	rGrossWeigth 	: LREAL;
	rNetWeigth		: LREAL;
	rNetVolume		: LREAL;
	rTargetVolume	: LREAL;
	rDifferencePercent	: LREAL;
	rDifferenceUl	: LREAL;
	rCriteria		: REAL;
	iPumpRevs		: UINT;
END_STRUCT
END_TYPE

// ---- DUTs/Calibration/ST_CalibrationInfo.TcDUT
TYPE ST_CalibrationInfo :
STRUCT
	iCalibrationNumber 	: UDINT;
	iUserID				: STRING(128);
	rSolventDensity 	: LREAL;
	iSolventID			: STRING(64);
	iSysMasterListRev 	: UDINT;
	iSysSettingsRev		: UDINT;
	iSolventRevision 	: UINT;
	iReplicates			: UINT;
	iAllowableFailures	: UINT;
	iCalIntervalDays	: UINT;
END_STRUCT
END_TYPE

// ---- DUTs/Calibration/ST_CalibrationPump.TcDUT
TYPE ST_CalibrationPump :
STRUCT
	bSelected       : BOOL;              // Se a bomba está selecionada para calibração
    rTargetVolume   : REAL;              // Volume desejado (em mL)
    rActualVolume   : REAL;              // Último volume medido (em mL)
    iFailures       : INT;               // Contador de falhas da bomba
    bAdjustment     : BOOL;              // Se um ajuste foi necessário
    eStatus         : E_CalibrationStatus; // Estado atual da bomba
    bBusy           : BOOL;              // Se a bomba está em operação
    tStartTime      : TIME;              // Timestamp do início da calibração
    tElapsed        : TIME;              // Tempo decorrido da calibração
END_STRUCT
END_TYPE

// ---- DUTs/Calibration/ST_CalibrationPumpResult.TcDUT
TYPE ST_CalibrationPumpResult :
STRUCT
	(* Pump Calibration screen controls feeding from FB_Calibration Manager *)
    rTargetVolume   : LREAL;              	// Target Volume 
    rAvgNetVolume   : LREAL;              	// Average Net Volume (mL)
	rAvgTareWeight	: LREAL;              	// Average Tare Weight (mg)
	rAvgGrossWeight	: LREAL;              	// Average Gross Weight(mg)
	iRevsDone		: UINT;            		// Number of revolutions done
    eStatus         : E_CalibrationStatus; 	// Actual pump calibration state
END_STRUCT
END_TYPE

// ---- DUTs/Calibration/ST_DosingResults.TcDUT
TYPE ST_DosingResults :
STRUCT
	iPump 		: USINT;
	iCheck		: USINT;
	rResult 	: LREAL;
	iRevs		: LREAL;
END_STRUCT
END_TYPE

// ---- DUTs/Calibration/ST_LinearPumpCalibration.TcDUT
TYPE ST_LinearPumpCalibration :
STRUCT
	bEnabled 		: BOOL;
	bHomed			: BOOL;
	rOldPosition	: LREAL;
	rNewPosition	: LREAL;
	rPumpFactor		: LREAL;
	bActivate		: BOOL;
END_STRUCT
END_TYPE

// ---- DUTs/Calibration/ST_LinearPumpControllDB.TcDUT
TYPE ST_LinearPumpControllDB :
STRUCT
	sPumpNumber		: STRING(2); 
	sOldPosition	: STRING(8);
	sNewPosition	: STRING(8);
	sUserName		: STRING(64);
	sDateOfChange	: STRING(64);
END_STRUCT
END_TYPE

// ---- DUTs/Calibration/ST_ReportInfo.TcDUT
TYPE ST_ReportInfo :
STRUCT
	sReportName		: STRING(256); 
    sReoportSubName	: STRING(256);
    sReportDate		: STRING(32);	
    sSystemID		: STRING(64);
    sDatabaseName 	: STRING(64);
    iPage			: USINT;
    sPrintedBy		: STRING(128);
END_STRUCT
END_TYPE

// ---- DUTs/Calibration/ST_ScaleReply.TcDUT
TYPE ST_ScaleReply :
STRUCT
	bOk        : BOOL;
    sRaw       : STRING(255);
    eKind      : (RespWeight, RespStatus, RespError, RespNone);
    cStatus    : STRING(1);     // 'S','D','A','B','L','I','+','-'
    rWeight    : LREAL;         // para SI/S/TA
    sUnit      : STRING(8);
END_STRUCT
END_TYPE

// ---- DUTs/HMI/E_IconState.TcDUT
{attribute 'qualified_only'}
{attribute 'strict'}
TYPE E_IconState :
(
	Waiting := 0,
	InProgress :=1,
	Completed := 2
);
END_TYPE

// ---- DUTs/HMI/ST_AX8101IOInfo.TcDUT
TYPE ST_AX8101IOInfo :
STRUCT
	bAxisOperational 	: BOOL;
	rActualPosition		: LREAL;
	rActualVelocity		: LREAL;
	rActualTorque		: LREAL;
	bAxisHomed			: BOOL;
	bNotMoving			: BOOL;
	bAxisError			: BOOL;
	bDriveError			: BOOL;
	nErrorCode			: UDINT;
END_STRUCT
END_TYPE

// ---- DUTs/HMI/ST_AMI8000IOInfo.TcDUT
TYPE ST_AMI8000IOInfo :
STRUCT
	bAxisOperational 	: BOOL;
	bNotMoving			: BOOL;
	rActualPosition		: LREAL;
	rActualVelocity		: LREAL;
	rActualTorque		: LREAL;
	bAxisHomed			: BOOL;
	bAxisError			: BOOL;
	nErrorCode			: UDINT;
END_STRUCT
END_TYPE

// ---- DUTs/HMI/ST_HMIAnimation.TcDUT
TYPE ST_HMIAnimation :
STRUCT
(*Here are all the variables needed to animate de HMI Controls.*)

//Level Sensors Animation
aSolventLevel	:	ARRAY[1..4] OF INT;
rWasteLevel		:	INT;

//Motors Position Animation
rM1VerticalAnimation	: REAL;
rM2VerticalAnimation	: REAL;

//Jars Animation
rJarFillAnimation : ARRAY[1..10] OF LREAL;

//Valvel Angles and Position Animation
aValveAngle		:	ARRAY[1..5] OF LREAL;
aValvePosition	:	ARRAY[1..5] OF INT;

//Rotary Pumps Animation
bPumpPositiveDirection	: ARRAY[1..10] OF BOOL;
bPumpNegativeDirection	: ARRAY[1..10] OF BOOL;

//Progress Circle Bar | Text | State Animation
rLoadBarSafety 	 : REAL;
rLoadBarAirFlow  : REAL;
rLoadBarSealing  : REAL;
rLoadBarHardware : REAL;
rLoadBarPrime  	 : REAL;
rLoadBarLeakTest : REAL;
rLoadBarRecovery : REAL;
rLoadBarWashing  : REAL;
rLoadBarDry 	 : REAL;

eIconStateSafety 	: E_IconState; 
eIconStateAirFlow 	: E_IconState;
eIconStateSealing 	: E_IconState;
eIconStateHardware 	: E_IconState;
eIconStatePrime 	: E_IconState;
eIconStateLeakTest 	: E_IconState;
eIconStateRecovery	: E_IconState;
eIconStateWashing 	: E_IconState;
eIconStateDry	 	: E_IconState;

sLoadTextSafety	 	: STRING(64);
sLoadTextAirFlow	: STRING(64);
sLoadTextSealing	: STRING(64);
sLoadTextHardware	: STRING(64);
sLoadTextPrime		: STRING(64);
sLoadTextLeakTest	: STRING(64);
sLoadTextRecovery	: STRING(64);
sLoadTextWashing	: STRING(64);
sLoadTextDry	 	: STRING(64);

//Doors hide/visible
bHMIDoorOpen	: ARRAY[1..6] OF BOOL;
bHMIDoorBlink	: ARRAY[1..6] OF BOOL;

//Pumping Flashing Arrows
aPumpingArrowFwd	: ARRAY[1..10] OF BOOL;
aPumpingArrowBwd	: ARRAY[1..10] OF BOOL;
 

END_STRUCT
END_TYPE

// ---- DUTs/HMI/ST_HMIDigInputs.TcDUT
TYPE ST_HMIDigInputs :
STRUCT	
	bRebootPLC				: BOOL := FALSE; //Reboot PLC bt from HMI
	bShutdownPLC			: BOOL := FALSE; //Shutdown PLC bt from HMI
END_STRUCT
END_TYPE

// ---- DUTs/HMI/ST_HMIDigOutputs.TcDUT
TYPE ST_HMIDigOutputs :
STRUCT
	bHMIResetButton	: BOOL; //Reset button light sent to HMI
	bHMIStartButton	: BOOL; //Start button light sent to HMI
	bHMIEStopSide	: BOOL; //Emergency stop button sent to HMI
	bHMIEStopFront	: BOOL; //Emergency stop button sent to HMI
	
	//Alarm Lamp HMI Indicators
	bAlarmLampRed	:	BOOL := FALSE;
	bAlarmLampAmbar	:	BOOL := FALSE;
	bAlarmLampGreen	:	BOOL := FALSE;
	
	
END_STRUCT
END_TYPE

// ---- DUTs/HMI/ST_HMIManual.TcDUT
TYPE ST_HMIManual :
STRUCT
	
END_STRUCT
END_TYPE

// ---- DUTs/HMI/ST_HMIParameters.TcDUT
TYPE ST_HMIParameters :
STRUCT
	
	tCheckAirFlowTime 	: TIME;				//Time in seconds to check air flow
	
	aM1Position : ARRAY [1..3] OF INT;		//M1 Motor - Stage Collection Vertical Axis  |1=HomePosition|2=SealPosition|3=DryPosition|
	aM2Position : ARRAY [1..6] OF INT;		//M2 Motor - Sample Recovery Vertical Axis   |1=HomePosition|2=IntoWaste|3=IntoVials|4=IntoResBottom|5=IntoResDispense|6=IntoResWeight|
	aM3Position : ARRAY [1..4] OF INT;		//M3 Motor - Sample Recovery Horizontal Axis |1=HomePosition/Waste|2=AboveVialSet1|3=VialsetSpacing|4=Calibration|
	fM1PositionDeceleration	: INT := 30;	//M1 Motor - the amount of mm to start the precision slow moviment to seal stages
	
	
	//Stage Collection Motor M1 - Vertical
	rM1Velocity			 :	LREAL;
	rM1PrecisionVelocity :	LREAL;
	rM1Accleration		 :	LREAL;
	rM1Deceleration		 :	LREAL;
	
	//Sample Recovey Motor M2 - Vertical
	rM2Velocity			 :	LREAL;
	rM2Accleration		 :	LREAL;
	rM2Deceleration		 :	LREAL;
	
	//Sample Recovey Motor M3 - Horizontal
	rM3Velocity			 :	LREAL;
	rM3Accleration		 :	LREAL;
	rM3Deceleration		 :	LREAL;


END_STRUCT
END_TYPE

// ---- DUTs/HMI/ST_InfoPage.TcDUT
TYPE ST_InfoPage :
STRUCT
	sApplication 	 : STRING(254);
	sProjectId		 : STRING(32);
	rSoftwareVersion : REAL;
	sTwincatVersion	 : STRING(254);
	sVSVersion		 : STRING(254);
	sDate			 : STRING(32);
END_STRUCT
END_TYPE

// ---- DUTs/HMI/ST_EL7062IOInfo.TcDUT
TYPE ST_EL7062IOInfo :
STRUCT
	bAxisOperational 	: ARRAY[1..2] OF BOOL;
	rActualPosition		: ARRAY[1..2] OF LREAL;
	rActualVelocity		: ARRAY[1..2] OF LREAL;
	rActualTorque		: ARRAY[1..2] OF LREAL;
	bAxisHomed			: ARRAY[1..2] OF BOOL;
	bAxisError			: ARRAY[1..2] OF BOOL;
	nErrorCode			: ARRAY[1..2] OF UDINT;
END_STRUCT
END_TYPE

// ---- DUTs/HMI/ST_MotorsJog.TcDUT
TYPE ST_MotorsJog :
STRUCT
	
	//Boolean variables linked to HMI for manual control of every 28 Axis in the project
	bMotorsJogFwd 		: ARRAY[1..3] OF BOOL;
	bMotorsJogBwd 		: ARRAY[1..3] OF BOOL;
	
	bValvesJogFwd 		: ARRAY[1..5] OF BOOL;
	bValvesJogBwd 		: ARRAY[1..5] OF BOOL;
		
	bPumpsLinearJogFwd 	: ARRAY[1..10] OF BOOL;
	bPumpsLinearJogBwd 	: ARRAY[1..10] OF BOOL;
		
	bPumpsRotaryJogFwd	: ARRAY[1..10] OF BOOL;
	bPumpsRotaryJogBwd	: ARRAY[1..10] OF BOOL;
	
END_STRUCT
END_TYPE

// ---- DUTs/HMI/ST_Reminders.TcDUT
TYPE ST_Reminders :
STRUCT
	bSolventLevels 		: BOOL := FALSE;
	bWasteLevel			: BOOL := FALSE;
	bVialRackPresent	: BOOL := FALSE;
	bRecipeActivated	: BOOL := FALSE;
	bThroatJigPresent	: BOOL := FALSE;
	bAutoCicleReady		: BOOL := FALSE;
	bStagePlateHomePos	: BOOL := FALSE;
	bVialRackRemoved	: BOOL := FALSE;
	bCalBoxInPlace		: BOOL := FALSE;
	bCalibrationReady	: BOOL := FALSE;
END_STRUCT
END_TYPE

// ---- DUTs/ifmLvlSensors/E_LevelSensorID.TcDUT
{attribute 'qualified_only'}
{attribute 'strict'}
TYPE E_LevelSensorID :
(
	Ch1_Rinse1 := 1,
    Ch2_Rinse2 := 2,
    Ch3_Rinse3 := 3,
    Ch4_Rinse4 := 4,
    Ch5_Waste  := 5
);
END_TYPE

// ---- DUTs/ifmLvlSensors/ST_KQ1000_Data.TcDUT
TYPE ST_KQ1000_Data :
STRUCT
	iRawLevel         : WORD;   // Raw Level (0–100 or 32764 = NoData)
    rLevelPercent     : REAL;   // % Level (0-100 or -1.0 para NoData)
    wStatusRaw        : WORD;   // Status complete word
    bOut1             : BOOL;   // Status OUT1
    bOut2             : BOOL;   // Status OUT2
    bOut3             : BOOL;   // Status OUT3
    iDeviceStatusCode : USINT;  // State Bits 4–7 
END_STRUCT
END_TYPE

// ---- DUTs/IO/ST_AL1333.TcDUT
TYPE ST_AL1333 :
STRUCT
	bStateIOLink				: ARRAY[1..8] OF BOOL;
	nStateIOLink		AT %I*	: ARRAY[1..8] OF USINT;
	bQualifierIOLink 			: ARRAY[1..8] OF BOOL;
	nQualifierIOLink 	AT %I*	: ARRAY[1..8] OF USINT;
END_STRUCT
END_TYPE

// ---- DUTs/IO/ST_AX8108.TcDUT
TYPE ST_AX8108 EXTENDS ST_Motor :
STRUCT
	//Terminal 45 AX8108-0100-0000	| Servomotor Driver with FSoE SS1 and STO, (Axis 1)
	//M1 Motor Stage Collection Vertical Axis
	
		
	//M1 Motor Safety
	bTS_Run				AT %Q*		: BOOL;
	bTS_ErrorAck		AT %Q*		: BOOL;
	
	//New variables
	rHomeVel      : LREAL;   // Homing Speed
	rHomeAcc	  : LREAL;   // Homing Acceleration	
	rHomeDec	  : LREAL;   // Homing Speed Deceleration
    rTargetPos    : LREAL;   // Absolute target position
    rTargetVel    : LREAL;   // Absolute target speed
    rAcceleration : LREAL;   // Default Acceleration for movements
    rDeceleration : LREAL;   // Default Deceleration for movements
	
END_STRUCT
END_TYPE

// ---- DUTs/IO/ST_EL1809.TcDUT
TYPE ST_EL1809 :
STRUCT
	
	//Terminal 9
	bStartButton 										: BOOL;  // Term9_I.1 Start Button 
    bStopButton 										: BOOL;  // Term9_I.2 Stop Button 
    b24VPowerSupplyOK 									: BOOL;  // Term9_I.3 24V Power Supply OK 
    b24VPowerSupplyOKBck 								: BOOL;  // Term9_I.4 24V Power Supply OK Backup 
    b48VPowerSupplyOK 									: BOOL;  // Term9_I.5 48V Power Supply OK 
    bStageCollection_Home 								: BOOL;  // Term9_I.6 Stage Collection Home Position 
    bSampleRecovery_Vertical_Home 						: BOOL;  // Term9_I.7 Sample Recovery Vertical Home 
    bSampleRecovery_Horizontal_Home 					: BOOL;  // Term9_I.8 Sample Recovery Horizontal Home 
    bWasteOverflowSensor 								: BOOL;  // Term9_I.9 Waste Overflow Sensor 
    bUPSReady 											: BOOL;  // Term9_I.10 UPS Ready 
    bUPSReplaceBattery 									: BOOL;  // Term9_I.11 UPS Replace Battery 
    b48VPowerSupplyOKBck 								: BOOL;  // Term9_I.12 48V Us Power Supply OK 
    bCalibrationBoxPresent 								: BOOL;  // Term9_I.13 Calibration Box Present 
    bThroatJigPresent 									: BOOL;  // Term9_I.14 Throat Jig Present 

	//Terminal 30
	bAccessDoor4InterlockFdbk							: BOOL;  // Term30_I.1 Keyence Access Door Interlock Feedback
	bAccessDoor5InterlockFdbk							: BOOL;  // Term30_I.1 Keyence Access Door Interlock Feedback
	bAccessDoor6InterlockFdbk							: BOOL;  // Term30_I.1 Keyence Access Door Interlock Feedback

END_STRUCT
END_TYPE

// ---- DUTs/IO/ST_EL2624.TcDUT
TYPE ST_EL2624 :
STRUCT
	//4-channel relay output / Lamps
	
	bStageCollectionLeftLight	:	BOOL; 	//Channel 1 - Stage Collection Left Side LED 
	bSampleRecoveryLight		:	BOOL;	//Channel 2 - Sample Recovery LED
	bStageCollectionRightLight	:	BOOL;	//Channel 3 - Stage Collection Right Side LED 
	
END_STRUCT
END_TYPE

// ---- DUTs/IO/ST_EL2809.TcDUT
TYPE ST_EL2809 :
STRUCT
	bStartIndicator 			: BOOL;  // Start Indicator 
    bResetIndicator 			: BOOL;  // Reset Indicator 
    bTowerRedLight 				: BOOL;  // Alarm Red Light 
    bTowerAmberLight 			: BOOL;  // Warning Amber Light 
    bTowerGreenLight	 		: BOOL;  // Auto Cycle Green Light 
    bTowerBuzzer 				: BOOL;  // Buzzer 
    bSolenoidValveB 			: BOOL;  // Solenoid Valve B 
    bSolenoidValveA 			: BOOL;  // Solenoid Valve A 
    bSolenoidValveC 			: BOOL;  // Solenoid Valve C 

END_STRUCT
END_TYPE

// ---- DUTs/IO/ST_EL3058.TcDUT
TYPE ST_EL3058 :
STRUCT
	//FESTO Main Air Pressure Supply Indicator
	rMainPressureSupplyInput 		: INT;  	// Main Pressure Supply (*AT I1*)
	bMainPressureSupplyError		: BOOL;		// Main Pressure Supply Error Status
	
	//SMC Pressure Regulator [Leak Detection]
    rPressureRegulatorInput			: INT;  	// Pressure Regulator (*AT I3*)
	bPressureRegulatorError			: BOOL;		// Pressure Regulator Error Status
	
	//2-channel analog input
	rLeakTestPressureSensor	:	INT; 	//SMC low differential pressure sensor (*AT I2*)
	bLeakTestSensorError	:	BOOL;	//SMC low differential pressure sensor Error Flag
	
END_STRUCT
END_TYPE

// ---- DUTs/IO/ST_EL6631.TcDUT
TYPE ST_EL6631 :
STRUCT
	bCurrentValueInvalid	: BOOL;
	bCurrentValueUnerRange	: BOOL;
	bCurrentValueOverRange	: BOOL;
	bWarningStatus			: BOOL;
	bErrorStatus			: BOOL;
	iCurrentValue			: DINT;
	iPnIoBoxState			: UINT;
END_STRUCT
END_TYPE

// ---- DUTs/IO/ST_EL6910.TcDUT
TYPE ST_EL6910 :
STRUCT
	// TERMINAL - EL6910 EtherCAT Coupler (Term 3)
	qSafetyRun                          	AT %Q*          :   BOOL;  	// Terminal 3 Start Safety
	qSafetyErrorAck							AT %Q* 			: 	BOOL;	// Terminal 3 Safety Acknowl
	iSafetyFBError	 						AT %I*			: 	BOOL;	// Terminal 3 At least one FB is in error condition
	qLockDoorsCommand						AT %Q*			:	BOOL;	// Terminal 3 Unlock all dors command
	qSafetyAirPresureOK                     AT %Q*          :   BOOL;   // Terminal 3 Safety Air Presure Check
	iSafetyRunning                          AT %I*          :   BOOL;   // Terminal 3 TwinSAFE running
	iSafetyComError 						AT %I*	 		: 	BOOL;	// Terminal 3 Communication error
	iSafetyOutError				     		AT %I*			:	BOOL;	// Terminal 3 Some other TwinSAFE error
	iSafetyOK								AT %I*			:	BOOL;	// Terminal 3 Safety outputs active - all safety gear OK
	iBypassDoor3Command						AT %I*			:	BOOL;	// Terminal 3 Safety inputs Alias bypass door 3
	nEL6910State							AT %I*			:	UINT;	// EL6910 State from IO Terminal Info Data	
	bEL6910State							AT %I*			:	BOOL;	// EL6910 State from IO Terminal Info Data	
	sEL6910Status											:	STRING(200);
END_STRUCT
END_TYPE

// ---- DUTs/IO/ST_EL7062.TcDUT
TYPE ST_EL7062 :
STRUCT
	//EtherCAT Terminal, 2-channel motion interface, stepper motor, 48 V DC
	Linear	:	ST_EL7062A1; //Axis 1 - Linear Pump 1 Amp (4600 steps limit)
	Rotary	:	ST_EL7062A2; //Axis 2 - Rotary pump 2 Amp (relative motion)
END_STRUCT
END_TYPE

// ---- DUTs/IO/ST_EL7062A1.TcDUT
TYPE ST_EL7062A1 EXTENDS ST_Motor :
STRUCT
	//Axis 1 - Pump Linear Actuator - 1A
	rHomeVel      : LREAL;   // Homing Speed
	rHomeAcc	  : LREAL;   // Homing Acceleration	
	rHomeDec	  : LREAL;   // Homing Speed Deceleration
    rTargetPos    : LREAL;   // Absolute target position
    rTargetVel    : LREAL;   // Absolute target speed
    rAcceleration : LREAL;   // Default Acceleration for movements
    rDeceleration : LREAL;   // Default Deceleration for movements
	
	//Terminal 23 to 32 - EL7062 UINT Input
	iHomeSensor	  	AT%I*   : UINT;
	bHomeSensorState   		: BOOL;
	
	(* 
	Manufactor Info 
	
	The movement OF the linear actuator is linear, meaning each step changes the 
	dispense volume BY a consistent amount. THIS volume change per step varies with 
	the piston size, as listed below: 

	- 3/16” – 0.013 µL/step  
	- 1/4”  – 0.037 µL/step  
	- 9mm   – 0.079 µL/step 
	*)

END_STRUCT
END_TYPE

// ---- DUTs/IO/ST_EL7062A2.TcDUT
TYPE ST_EL7062A2 EXTENDS ST_Motor :
STRUCT
	//Axis 2 - Pump Rotary Actuator - 2A
	nStepsPerRev			: UDINT := 200;		// Number of steps per revolution
    nCurrentStep  			: DINT;   			// Current Step
    rSpeed        			: REAL;   			// Current Velocity (RPM)
	rDistance     			: LREAL; 			// Relative distance to be moved (Steps)
    rRelVelocity  			: REAL := 1000;  	// Relative Velocity
    rAcceleration 			: REAL := 1500; 	// Acceleration for relative motion
	rDeceleration			: REAL := 1500;		// Deceleration for relative motion
	rPumpFactorFillJars		: LREAL; 			// the ratio between degrees/setps and volume by path - from solvent botles to jars
	rPumpFactorFillCalBox	: LREAL; 			// the ratio between degrees/setps and volume by path - from jars to calibration box
	rPumpFactorFromCalBox	: LREAL; 			// the ratio between degrees/setps and volume by path - from calibration box to the jars
	rDeadVolume				: REAL;				// Dead Volume in the pipes to be added to the volume pumping
END_STRUCT
END_TYPE

// ---- DUTs/IO/ST_EL7211.TcDUT
TYPE ST_EL7211 EXTENDS ST_Motor :
STRUCT
	
	//Terminals 27 n 28 EL7211-9014	| Servomotor Terminal with OCT and STO, 48 V (Axis 1)
	//M2 and M3 Motors Stage collection matrix Axis
	
	//New variables
	rHomeVel      : LREAL;   // Homing Speed
	rHomeAcc	  : LREAL;   // Homing Acceleration	
	rHomeDec	  : LREAL;   // Homing Speed Deceleration
	rTargetPos    : LREAL;   // Absolute target position
	rTargetVel    : LREAL;   // Absolute target speed
	rAcceleration : LREAL;   // Default Acceleration for movements
	rDeceleration : LREAL;   // Default Deceleration for movements
	
END_STRUCT
END_TYPE

// ---- DUTs/IO/ST_EP9208.TcDUT
TYPE ST_EP9208 EXTENDS ST_Motor :
STRUCT
	//VICI Valves connected to EP9208-1035
	
	//New Variables
	rHomeVel      : LREAL;   // Homing Speed
	rHomeAcc	  : LREAL;   // Homing Acceleration	
	rHomeDec	  : LREAL;   // Homing Speed Deceleration
    rTargetPos    : LREAL;   // Absolute target position
    rTargetVel    : LREAL;   // Absolute target speed
    rAcceleration : LREAL;   // Default Acceleration for movements
    rDeceleration : LREAL;   // Default Deceleration for movements
	
END_STRUCT
END_TYPE

// ---- DUTs/ManualControl/E_SolenoidSet.TcDUT
{attribute 'qualified_only'}
{attribute 'strict'}
TYPE E_SolenoidSet :
(
	IDLE 				:= 1,	//Idle position all solenoids in false
    LEAKTEST 			:= 2,	//Leak Test position
    LEAKTESTMONITORING 	:= 3,	//Leak Test monitoring position
    AIRDRY 				:= 4 	//air dry position
);
END_TYPE

// ---- DUTs/ManualControl/ST_MotorCommand.TcDUT
TYPE ST_MotorCommand :
STRUCT
	bRun         : BOOL;
    bStop        : BOOL;
    iPosition    : INT;
    bBusy        : BOOL;
END_STRUCT
END_TYPE

// ---- DUTs/ManualControl/ST_PumpCommand.TcDUT
TYPE ST_PumpCommand :
STRUCT
	bRunBySpeed  : BOOL;
    bRunByVolume : BOOL;
    bStop        : BOOL;
    bActive      : BOOL;
    eDirection   : E_PumpDirection;
    rSpeed       : REAL; // % or RPM
    rVolume      : REAL; // mL or user unit
	iDistance	 : UINT; // Revs number
    bBusy        : BOOL;
END_STRUCT
END_TYPE

// ---- DUTs/ManualControl/ST_ValveCommand.TcDUT
TYPE ST_ValveCommand :
STRUCT
	bMove        : BOOL;
    bStop        : BOOL;
    iTargetPos   : USINT; // 1..6
    bBusy        : BOOL;
END_STRUCT
END_TYPE

// ---- DUTs/MotionControl/E_ActuatorState.TcDUT
{attribute 'qualified_only'}
{attribute 'strict'}
TYPE E_ActuatorState :
(
	eIdle,
    eActive,
    eDisabled,
    eError
);
END_TYPE

// ---- DUTs/MotionControl/E_MotorType.TcDUT
{attribute 'qualified_only'}
{attribute 'strict'}
TYPE E_MotorType :
(
	eLinear,
    eRotary,
    eStepper
);
END_TYPE

// ---- DUTs/MotionControl/E_PumpPath.TcDUT
{attribute 'qualified_only'}
{attribute 'strict'}
TYPE E_PumpPath :
(
    FillJars   := 0, 	// From solvent bottles to jars
    FillCalBox := 1, 	// From jars to calibration box
    FromCalBox := 2 	// From calibration box to the jars
) UDINT;
END_TYPE

// ---- DUTs/MotionControl/ST_ActuatorStatus.TcDUT
TYPE ST_ActuatorStatus :
STRUCT
	bEnabled    : BOOL;
    bBusy       : BOOL;
    bDone       : BOOL;
    bError      : BOOL;
    iErrorCode  : UDINT;
    fPosition   : LREAL;
	bMovingFwd	: BOOL;
	bMovingBck	: BOOL;
    eState      : E_ActuatorState;
    sMessage    : STRING[80];	
END_STRUCT
END_TYPE

// ---- DUTs/MotionControl/ST_AxisReadStatus.TcDUT
TYPE ST_AxisReadStatus :
STRUCT
	//Some Status from MC_ReadStatus
	Disabled 			: BOOL;
	Error 				: BOOL;
	ErrorID 			: UDINT;
	Homed 				: BOOL;
	Operational 		: BOOL;
	StandStill 			: BOOL;
	MotionCommandsLocked : BOOL;
END_STRUCT
END_TYPE

// ---- DUTs/MotionControl/ST_Motor.TcDUT
TYPE ST_Motor :
STRUCT
	Axis        : AXIS_REF;   // Axis reference (default to all motors)
    bEnable     : BOOL;       // Enable command
    bReset      : BOOL;       // Reset command
    bError      : BOOL;       // Error flag
    nErrorID    : UDINT;      // Error ID
    bBusy       : BOOL;       // In moviment state
    bInPosition : BOOL;       // Indicates when the position was reached
	rActualPosition : LREAL;  // Show de actual motor position
	
	// Additional variables to direct link (%I e %Q):
    nState        	AT %I*	: UINT;	 //Actual State (Axis StatusWord)
    nControlWord  	AT %Q*	: UINT;	 //Control Word (ControlWord send to axis)
    rActualPos 		AT %I*	: LREAL; //Real Actual Axis Position (Position Actual Value)
	rActualTorque	AT %I*	: LREAL; //Real Actual Axis Torque (Torque Actual Value)
    rActualVel 		AT %I*	: LREAL; //Real Actual Axis Velocity (Velocity Actual Value)
	iOperational	AT %I*	: BOOL;
	iHomed			AT %I*	: BOOL;
	iNotMoving		AT %I*	: BOOL;
	iError			AT %I*	: BOOL;
	nErrorCode		AT %I*	: UDINT;
	bMotionCommandsLocked	AT %I*	: BOOL;
	bPositiveDirection		AT %I*	: BOOL;
	bNegativeDirection		AT %I*	: BOOL;
	
END_STRUCT
END_TYPE

// ---- DUTs/MotionControl/ST_SolenoidSet.TcDUT
TYPE ST_SolenoidSet :
STRUCT
	
	bSolenoidA 		: BOOL;  // Solenoid Valve A
    bSolenoidB 		: BOOL;  // Solenoid Valve B 
    bSolenoidC 		: BOOL;  // Solenoid Valve C 
	
END_STRUCT
END_TYPE

// ---- DUTs/Recipe/ST_HMI_OtherParamsRow.TcDUT
TYPE ST_HMI_OtherParamsRow :
STRUCT
	Parameter : STRING(32);
    Value     : REAL;
    Units     : STRING(8);
END_STRUCT
END_TYPE

// ---- DUTs/Recipe/ST_HMI_SolventAndTimeRow.TcDUT
TYPE ST_HMI_SolventAndTimeRow  :
STRUCT
	Parameter : STRING(16);
    Rinse1    : INT;
    Rinse2    : INT;
    Wash1     : INT;
    Wash2     : INT;
END_STRUCT
END_TYPE

// ---- DUTs/Recipe/ST_HMI_VolumesRow.TcDUT
TYPE ST_HMI_VolumesRow  :
STRUCT
	Stage  : STRING(8);     // "T/IC", "S0", ..., "F"
    Rinse1 : REAL;
    Rinse2 : REAL;
    Wash1  : REAL;
    Wash2  : REAL;
END_STRUCT
END_TYPE

// ---- DUTs/Recipe/ST_Recipe.TcDUT
TYPE ST_Recipe :
STRUCT
    stInfo           : ST_RecipeInfo;
    stSolventsTimes  : ST_RecipeSolventAndTimes;
    stVolumes        : ST_RecipeVolumes;
    stOtherParams    : ST_RecipeOtherParams;
END_STRUCT
END_TYPE

// ---- DUTs/Recipe/ST_RecipeFileInfo.TcDUT
TYPE ST_RecipeFileInfo :
STRUCT
	sFileName      : STRING(128); 	// Nome do arquivo .json
    dtLastModified : DT;         	// Timestamp do arquivo
    sCreatedBy     : STRING(64); 	// From JSON
    dCreationDate  : DATE;       	// From JSON
	sMethodName	   : STRING;  		// From JSON
    iRevision      : INT;        	// From JSON
END_STRUCT
END_TYPE

// ---- DUTs/Recipe/ST_RecipeInfo.TcDUT
TYPE ST_RecipeInfo :
STRUCT
	//Info Group 
	sMethodName			: STRING;  	//Method/Recipe Name
	iRevision			: INT; 		//Revision Number
	sCreatedBy			: STRING;  	//Name of the person responsible for the recipe creation
	dCreationDate		: DATE; 	//Recipe creation date
END_STRUCT
END_TYPE

// ---- DUTs/Recipe/ST_RecipeOtherParams.TcDUT
TYPE ST_RecipeOtherParams :
STRUCT
	//Other Parameters Group 
	tSoakTime 			: TIME; 	//Time in seconds for the soak step 
	tAgitate1Time 		: TIME; 	//Time in seconds for the Rinse 1 recirculation  
	tAgitate2Time 		: TIME; 	//Time in seconds for the Rinse 1 recirculation   
	iVialsToFill 		: USINT; 	//number 1 to 4 meaning the quantity of Vials line to be filled
	rVialPrimeVol 		: REAL; 	//Volume to be wasted in the prime needle
	rVial1FillVol 		: REAL; 	//Volume used to fill up the first line vials 
	rVials2_4FillVol 	: REAL; 	//Volume used to fill up the second up to fourth line vials 
	tAirDryTime 		: TIME; 	//Time in seconds in the dry step
END_STRUCT
END_TYPE

// ---- DUTs/Recipe/ST_RecipeSolventAndTimes.TcDUT
TYPE ST_RecipeSolventAndTimes :
STRUCT
	//Solvent AND Times Group [1..4] |Rinse 1|Rinse 2|Wash 1| Wash 2| 
	aSolventN 			: ARRAY [1..4] OF USINT; //Solvent number to be used on Rinse 1 | Rinse 2 | Wash 1 | Wash 2 
	aTime 				: ARRAY [1..4] OF TIME;  //time in seconds for each step Rinse 1 | Rinse 2 | Wash 1 | Wash 2 
	aVelocity 			: ARRAY [1..4] OF INT; 	 //rpm number for each step Rinse 1 | Rinse 2 | Wash 1 | Wash 2 
END_STRUCT
END_TYPE

// ---- DUTs/Recipe/ST_RecipeVolumes.TcDUT
TYPE ST_RecipeVolumes :
STRUCT
	//Volumes Group [1..4] |Rinse 1|Rinse 2|Wash 1| Wash 2| 
	aT_IC_Volume 		: ARRAY [1..4] OF REAL; //T/IC Solvent Volume for each step Rinse 1 | Rinse 2 | Wash 1 | Wash 2 
	aS0_Volume 			: ARRAY [1..4] OF REAL; //S0 Solvent Volume for each step Rinse 1 | Rinse 2 | Wash 1 | Wash 2 
	aS1_Volume 			: ARRAY [1..4] OF REAL; //S1 Solvent Volume for each step Rinse 1 | Rinse 2 | Wash 1 | Wash 2 
	aS2_Volume 			: ARRAY [1..4] OF REAL; //S2 Solvent Volume for each step Rinse 1 | Rinse 2 | Wash 1 | Wash 2 
	aS3_Volume 			: ARRAY [1..4] OF REAL; //S3 Solvent Volume for each step Rinse 1 | Rinse 2 | Wash 1 | Wash 2 
	aS4_Volume 			: ARRAY [1..4] OF REAL; //S4 Solvent Volume for each step Rinse 1 | Rinse 2 | Wash 1 | Wash 2 
	aS5_Volume 			: ARRAY [1..4] OF REAL; //S5 Solvent Volume for each step Rinse 1 | Rinse 2 | Wash 1 | Wash 2 
	aS6_Volume 			: ARRAY [1..4] OF REAL; //S6 Solvent Volume for each step Rinse 1 | Rinse 2 | Wash 1 | Wash 2 
	aS7_Volume 			: ARRAY [1..4] OF REAL; //S7 Solvent Volume for each step Rinse 1 | Rinse 2 | Wash 1 | Wash 2 
	aF_Volume 			: ARRAY [1..4] OF REAL; //F  Solvent Volume for each step Rinse 1 | Rinse 2 | Wash 1 | Wash 2 
END_STRUCT
END_TYPE

// ---- DUTs/Report/ST_CalibHeaderTest.TcDUT
{attribute 'pack_mode' := '1'}
TYPE ST_CalibHeaderTest :
STRUCT
    sCalibrationNo : STRING(30);
    sUserId        : STRING(50);
END_STRUCT
END_TYPE

// ---- DUTs/Report/E_ReportType.TcDUT
{attribute 'qualified_only'}
{attribute 'strict'}
TYPE E_ReportType :
(
	None := 0,
    PumpCalibration := 1,
    SystemSettings := 2,
    PostRun := 3,
    LinearMotors := 4,
    Recipe := 5
);
END_TYPE

// ---- DUTs/Report/ST_CompleteMethodHeader.TcDUT
TYPE ST_CompleteMethodHeader :
STRUCT
    methodName          : STRING(100);
    methodRevision      : STRING(100);
    methodCreatedBy     : STRING(100);
    methodCreatedOn     : STRING(100);
    solvent_R1          : STRING(100);
    solvent_R2          : STRING(100);
    solvent_W1          : STRING(100);
    solvent_W2          : STRING(100);
    time_R1             : STRING(100);
    time_R2             : STRING(100);
    time_W1             : STRING(100);
    time_W2             : STRING(100);
    velocity_R1         : STRING(100);
    velocity_R2         : STRING(100);
    velocity_W1         : STRING(100);
    velocity_W2         : STRING(100);
    soakTime            : STRING(100);
    agitate_1_Time      : STRING(100);
    agitate_2_Time      : STRING(100);
    vialsToFill         : STRING(100);
    vialPrimeVol        : STRING(100);
    vial_1_FillVol      : STRING(100);
    vial_2_4_FillVol    : STRING(100);
    airDryTime          : STRING(100);
    methodID            : INT;
    methodStatus        : STRING(100);
END_STRUCT
END_TYPE

// ---- DUTs/Report/ST_LinearReport.TcDUT
TYPE ST_LinearReport :
STRUCT
	ID_Linear  : INT;
    pump1      : STRING(100);
    pump2      : STRING(100);
    pump3      : STRING(100);
    pump4      : STRING(100);
    pump5      : STRING(100);
    pump6      : STRING(100);
    pump7      : STRING(100);
    pump8      : STRING(100);
    pump9      : STRING(100);
    pump10     : STRING(100);
    changedBy  : STRING(100);
    changedOn  : STRING(100);
END_STRUCT
END_TYPE

// ---- DUTs/Report/ST_ReportListItem.TcDUT
{attribute 'pack_mode' := '1'}
TYPE ST_ReportListItem :
STRUCT
	ReportType  : STRING(50);    // Ex: Pump Calibration, System Settings, Post Run
    ReportID    : STRING(50);    // Ex: CalibrationNo, RunID, Revision
    CreatedOn   : STRING(30);    // Ex: 2026-04-15 10:35
    CreatedBy   : STRING(50);    // Ex: Renan, Admin
    Description : STRING(200);   // Ex: Pump 3 calibration - Solvent 2
	sPrimaryKey : STRING(50);
END_STRUCT
END_TYPE

// ---- DUTs/Report/ST_ReportListItem_Test.TcDUT
{attribute 'pack_mode' := '1'}
TYPE ST_ReportListItem_Test :
STRUCT
    ReportType : STRING(50);
    ReportID   : STRING(50);
	CreatedOn  : STRING(30);
	CreatedBy  : STRING(50);
	Description : STRING(200);
	sPrimaryKey : STRING(50);
END_STRUCT
END_TYPE

// ---- DUTs/Report/ST_ReportPostRun.TcDUT
TYPE ST_ReportPostRun :
STRUCT
    sPrintGeneratedBy : STRING(50); // Name of the operator who triggered the PDF generation (optional)

    dtExecutionStart  : DT; // Date and time when the ASRS run started
    dtExecutionEnd    : DT; // Date and time when the ASRS run completed

    sMethodName       : STRING(100); // Name of the method/recipe executed
    iMethodRevision   : INT; // Revision number of the method
    sCreatedBy        : STRING(50); // User who originally created the method
    dtCreatedOn       : DT; // Date and time when the method was created

    aSolventNumber    : ARRAY[1..4] OF INT; // Solvent index used in each step
    aStepTime_sec     : ARRAY[1..4] OF INT; // Step duration in seconds
    aStepRPM          : ARRAY[1..4] OF INT; // RPM used in each step

    rSoakTime_sec     : REAL; // Soaking time in seconds
    rAgitate1Time_sec : REAL; // Agitation phase 1 duration in seconds
    rAgitate2Time_sec : REAL; // Agitation phase 2 duration in seconds
    iVialsToFill      : INT;  // Number of vials to fill
    rVialPrimeVol_ml  : REAL; // Volume used to prime the vial in milliliters
    rVial1FillVol_ml  : REAL; // Fill volume for the first vial in milliliters
    rVials2to4FillVol_ml : REAL; // Fill volume for vials 2 to 4 in milliliters
    rAirDryTime_sec   : REAL; // Air drying time in seconds

    aVolumeData : ARRAY[1..10] OF ST_VolumeLine; // Volume information for each pump/stage

    sAnalystName  : STRING(50); // Name of the analyst who ran the sample
    iRunNumber    : DINT; // Unique identifier for the run
    iCalibrationNumber : DINT; // Calibration number used during the run
    sComment      : STRING(100); // Optional comment about the run

    sSoftwareVersion : STRING(20); // Software version of the ASRS system
    iMasterRevision  : INT; // Master configuration revision
    iSettingsRevision : INT; // System settings revision
    iMeterVelocityRPM : INT; // Velocity for metering flow, in RPM
    iRunVelocityRPM   : INT; // Runtime velocity, in RPM
    rEmptyTubesFactor_ml : REAL; // Calibration factor for empty tubes in milliliters
    rFillTubesFactor_ml  : REAL; // Calibration factor for filled tubes in milliliters

    aSolvents : ARRAY[1..4] OF ST_SolventInfo; // Detailed solvent information used in the run
    aEvents   : ARRAY[1..10] OF ST_RunEvent; // Chronological list of events (start, complete, etc.)
END_STRUCT
END_TYPE

// ---- DUTs/Report/ST_RunEvent.TcDUT
TYPE ST_RunEvent :
STRUCT
    dtTimestamp : DT; // Timestamp of the event (e.g., start, end)
    sEvent      : STRING(50); // Description of the event (e.g., "Started", "Completed")
END_STRUCT
END_TYPE

// ---- DUTs/Report/ST_SolventInfo.TcDUT
TYPE ST_SolventInfo :
STRUCT
    sName     : STRING(50); // Name of the solvent (e.g., Water, Methanol)
    iRevision : INT; // Revision/version of the solvent definition
END_STRUCT
END_TYPE

// ---- DUTs/Report/ST_SystemSettingsReport.TcDUT
{attribute 'pack_mode' := '1'}
TYPE ST_SystemSettingsReport :
STRUCT
	sGenSealAndPump               : STRING(100);
    sCalAcceptanceCriteria        : STRING(100);
    sCalAllowableFail             : STRING(100);
    sCalReplicates                : STRING(100);
    sCalPumpCallIntervalDays      : STRING(100);
    sCalCloseAppOnCompletion      : STRING(100);
    sAirDryTimeOnCompletion       : STRING(100);
    sLktAllowableLeakTestFail     : STRING(100);
    sLktLeakTestBuildUpTime       : STRING(100);
    sLktLeakTestHoldTime          : STRING(100);
    sLktLeakTestPressure          : STRING(100);
    sMecPlatesClosedPosition      : STRING(100);
    sMecPlatesDryPosition         : STRING(100);
    sMecPlatesVelocity            : STRING(100);
    sMecMaxCurrentFastDown        : STRING(100);
    sMecMaxCurrentSlowDown        : STRING(100);
    sMecMaxCurrentSlowUp          : STRING(100);
    sPmpMeterVelocity             : STRING(100);
    sPmpRunVelocity               : STRING(100);
    sPmpEmptyFactor               : STRING(100);
    sPmpFillSolventTubesFactor    : STRING(100);
    sSmpAboveCalibration          : STRING(100);
    sSmpVialSetSpacing            : STRING(100);
    sSmpIntoResBottom             : STRING(100);
    sSmpIntoResDispense           : STRING(100);
    sSmpIntoResWeigh              : STRING(100);
    sSmpIntoVials                 : STRING(100);
    sSmpIntoWaste                 : STRING(100);
    sSecDisplayManualControl      : STRING(100);
    sSecCheckLogonEachRun         : STRING(100);
    sCreatedBy                    : STRING(100);
    sCreatedDate                  : STRING(100);
    sSysRevisionNo                : STRING(30);
END_STRUCT
END_TYPE

// ---- DUTs/Report/ST_VolumeLine.TcDUT
TYPE ST_VolumeLine :
STRUCT
    iPump   : INT; // Pump number (1 to 10)
    sStage  : STRING(10); // Stage name or ID (e.g., S0, S1, Cone)
    rRinse1 : REAL; // Volume used in Rinse 1 phase for this stage (ml)
    rRinse2 : REAL; // Volume used in Rinse 2 phase for this stage (ml)
    rWash1  : REAL; // Volume used in Wash 1 phase for this stage (ml)
    rWash2  : REAL; // Volume used in Wash 2 phase for this stage (ml)
END_STRUCT
END_TYPE

// ---- DUTs/Safety/ST_SafetyInputs.TcDUT
TYPE ST_SafetyInputs :
STRUCT
	//Term 16 EL1918
	bEStopHMICh1				:	BOOL; //I1 - Front eStop button channel 1
	bEStopHMICh2				:	BOOL; //I2 - Front eStop button channel 1
	bEStopSideCh1				:	BOOL; //I3 - Side eStop button channel 1
	bEStopSideCh2				:	BOOL; //I4 - Side eStop button channel 2
	bMachineReset				:	BOOL; //I5 - Reset Button
	bStageCollectLeftDoorCh1	:	BOOL; //I6 - D1 Door mechanic sensor channel 1
	bStageCollectLeftDoorCh2	:	BOOL; //I7 - D1 Door mechanic sensor channel 2
	bStageCollectLeftDoorFdbk	:	BOOL; //I8 - D1 Door mechanic sensor Feedback Signal

	//Term 17 EL1918
	bStageCollectRightDoorCh1	:	BOOL; //D2 Door mechanic sensor channel 1
	bStageCollectRightDoorCh2	:	BOOL; //D2 Door mechanic sensor channel 2
	bStageCollectRightDoorFdbk	:	BOOL; //D2 Door mechanic sensor Feedback Signal
	bSampleRecoveryDoorCh1		:	BOOL; //D3 Door mechanic sensor channel 1
	bSampleRecoveryDoorCh2		:	BOOL; //D3 Door mechanic sensor channel 2
	bSampleRecoveryDoorFdbk		:	BOOL; //D3 Door mechanic sensor Feedback Signal

	//Term 18 EL1918
	bFestoMS6ValveFdbk			:	BOOL; //I1 - Feedback from Festo MS6 Valve
	bFestoMS6DumpValveFdbk		:	BOOL; //I2 - Feedback from Festo MS^ Dump Valve
	bD4AccessDoorIntlckOSSD1	: 	BOOL; //I3 - D4 Access Door Interlock - OSSD1
	bD4AccessDoorIntlckOSSD2  	:	BOOL; //I4 - D4 Access Door Interlock - OSSD2
	bD5AccessDoorIntlckOSSD1  	:	BOOL; //I5 - D5 Access Door Interlock - OSSD1
	bD5AccessDoorIntlckOSSD2  	:	BOOL; //I6 - D5 Access Door Interlock - OSSD2
	bD6AccessDoorIntlckOSSD1  	:	BOOL; //I7 - D5 Access Door Interlock - OSSD1
	bD6AccessDoorIntlckOSSD2  	:	BOOL; //I7 - D5 Access Door Interlock - OSSD2
	
	//Safety Messages and variables
	iSafetyFBError	 			: 	BOOL;	// Terminal EL6910 - At least one FB is in error condition
	iSafetyComError 			: 	BOOL;	// Terminal EL6910 - Communication error
	bSafetyError				:	BOOL	; //6910 system erro  	
	bSafetyAirError       		:	BOOL;	// fault message 
	bSafetyAirOK          		:	BOOL;	// 	
	bSafetyAirPressurising   	: 	BOOL;
	bSafety_AirNotON       		: 	BOOL;
	iSafetyRunning          	:	BOOL;   // Terminal EL6910 TwinSAFE running
    iSafetyEStop    	   		:	BOOL;   // Terminal EL6910 Safety Estop OK
	bSafetyEstopDoorOK			:	BOOL;	//(from 1091) doors locked so enable air reset  
	
	//Motors STO 
	bM1STOEnabled				:	BOOL;
	bM1_STOActive				:	BOOL;
	
	//3 safty card status	
	nEL6910_State				:	UINT;	// EL6910 State from IO Terminal Info Data	
	sEL6910_Status				:	STRING(200);

END_STRUCT
END_TYPE

// ---- DUTs/Safety/ST_SafetyOutputs.TcDUT
TYPE ST_SafetyOutputs :
STRUCT
	//Term 19 EL2904
	bStageCollectLeftDoorCtrlSignal		:	BOOL; //Q1 - D1 Door mechanic Stage Collection Control Signal
	bStageCollectRightDoorCtrlSignal	:	BOOL; //Q2 - D2 Door mechanic Stage Collection Control Signal
	bSampleRecoveryDoorCtrlSignal		:	BOOL; //Q3 - D3 Door mechanic Stage Collection Control Signal
	
	//Term 20 EL2904
	bM2MotorSTO							:	BOOL; //Q1 - STO Signal Motor M2
	bM3MotorSTO							:	BOOL; //Q2 - STO Signal Motor M3
	bAirSupplyUnitEnable				: 	BOOL; //Q3 - Air Supply Unity - Enable
	bAirSupplyUnitReset					: 	BOOL; //Q3 - Air Supply Unity - Reset
	
	//Term 15 EL6910 Safety PLC, Virtual Channels 
	qSafetyErrorAck						: 	BOOL;	// Terminal EL6910 - Safety Acknowl
	qSafetyRun                  		:   BOOL;  	// Terminal EL6910 - Start Safety
	bAirPressureOK						:	BOOL;	// Terminal EL6910 - Reading from the Festo pressure sensor above 4.5 bar
	bResetAir							:	BOOL;	// Terminal EL6910 - Reset available only when air pressure is off	
	bLockDoorSafety        				: 	BOOL;	// lock doors cmd to safety logic
	bBelowDoorsFeedback					:	BOOL;	// Feedback signal from doos D4, D5 and D6, going to alias input BelowDoorsFeedback
	
	bTrueVariable						:	BOOL := TRUE;

END_STRUCT
END_TYPE

// ---- DUTs/Settings/ST_CalibrationSettings.TcDUT
TYPE ST_CalibrationSettings :
STRUCT
	iAllowableFailures		: USINT;
	iReplicatesSetpoint		: UINT;
	rAcceptanceCriteria		: LREAL;
	iCalIntervalDays		: UINT;
	iAirDryTimeSec			: UINT;
	iDelayTimeMin         	: INT;   
	bDelayStart				: BOOL := FALSE;
	bPrintWhenComplete		: BOOL := FALSE;
END_STRUCT
END_TYPE

// ---- DUTs/Settings/ST_LeakTestSettings.TcDUT
TYPE ST_LeakTestSettings :
STRUCT
	iAllowableLeakTestFailures	: UINT := 2;	 // Allowable leak test failures
	tLeakTestBuildUpTime		: UINT := 10; 	 // Time to be pressuring up the system
	tLeakTestMonitorTime		: UINT := 5;	 // Time to hold and monitoring the pressure into the system
	rLeakTestPressureLimit		: REAL := 3.8;	 // Leak test pressure threshold 
END_STRUCT
END_TYPE

// ---- DUTs/Settings/ST_PumpSettings.TcDUT
TYPE ST_PumpSettings :
STRUCT
	iMeterVelocity			: UINT;
	iRunVelocity			: UINT;
	iEmptyFactor			: UINT;
	iFillolventTubesFactor	: UINT;
END_STRUCT
END_TYPE

// ---- DUTs/Settings/ST_SolventsSettings.TcDUT
TYPE ST_SolventsSettings :
STRUCT
	sSolventName	: STRING(80); 	// The name of the solvent inserted on the settings screen
	rDensity		: LREAL;		// The density of this solvent
END_STRUCT
END_TYPE

// ---- DUTs/UserManagement/E_UserGroup.TcDUT
{attribute 'qualified_only'}
{attribute 'strict'}
TYPE E_UserGroup :
(
	Admin := 0,
    Operator := 1,
    Guest := 2
);
END_TYPE

// ---- DUTs/UserManagement/ST_User.TcDUT
TYPE ST_User :
STRUCT
	sUsername            : STRING(50);
    sDisplayName         : STRING(100);
    sPasswordHash        : STRING(64); // SHA-256 ou similar
    eGroup               : E_UserGroup;
    dtCreated            : DT;
    sCreatedBy           : STRING(50);
    dtLastPasswordChange : DT;
    tAutoLogoutTime      : TIME;
    bBlocked             : BOOL;
    nFailedLoginCount    : UINT;
    bForcePasswordReset  : BOOL;
    stStats              : ST_UserStats;;
END_STRUCT
END_TYPE

// ---- DUTs/UserManagement/ST_UserStats.TcDUT
TYPE ST_UserStats :
STRUCT
	dtLastLogin         : DT;
    dtLastLogout        : DT;
    nLoginsSuccess      : UDINT;
    nLoginsFailed       : UDINT;
    nRecipesCreated     : UDINT;
    nRecipesEdited      : UDINT;
    nRecipesDeleted     : UDINT;
    nCalibrations       : UDINT;
    nAutomaticCyclesRun : UDINT;
    dtLastAutoCycle     : DT;
    tAverageSessionTime : TIME;
END_STRUCT
END_TYPE

// ---- DUTs/Utility/E_PowerAction.TcDUT
{attribute 'qualified_only'}
{attribute 'strict'}
TYPE E_PowerAction :
(
	NONE, 
	SHUTDOWN, 
	REBOOT
);
END_TYPE

// ---- DUTs/Utility/E_SeqState.TcDUT
{attribute 'qualified_only'}
{attribute 'strict'}
TYPE E_SeqState :
(
	STANDBY, 
	WRITE_REQ, 
	WRITE_WAIT, 
	COUNTDOWN, 
	EXECUTE
);
END_TYPE

// ---- POUs/MARCO/DB/STs/E_DB_QUERY_STATE.TcTLEO
{attribute 'qualified_only'}
{attribute 'strict'}
TYPE E_DB_QUERY_STATE :
(
	IDLE_STATE,
	SELECT_POST_LAST_RUN,
	INSERT_RUN,
	SELECT_LAST_CALIBRATION_ID,
	INSERT_CALIBRATION_VALUES,
	INSERT_CALIBRATION,
	SELECT_LAST_SYSTEM_ID,
	SELECT_ALL_SYSTEM,
	INSERT_SYS_PARAMETERS,
	SELECT_ALL_METHODS,
	SELECT_ALL_ACTV_METHODS,
	SELECT_WHOLE_METHODS,
	INSERT_NEW_METHOD,
	UPDATE_DEACTV_METHOD,
	SELECT_LAST_METHOD_ID,
	SELECT_VOLUME_DATA,
	INSERT_VOLUME_DATA,
	SELECT_ALL_CURRENT_USERS,
	SELECT_ALL_USERS,
	SELECT_LAST_SOLVENT,
	SELECT_ALL_SOLVENT,
	INSERT_SOLVENT,
	INSERT_LINEAR_MOTORS,
	SELECT_LINEAR_MOTORS,
	SELECT_LAST_CALIBRATION,
	SELECT_CALIB_REPORT_LIST,
	SELECT_CALIB_REPORT_DETAILS,
	SELECT_SYSTEM_REPORT_LIST,
	SELECT_SYSTEM_REPORT_DETAILS,
	SELECT_POSTRUN_REPORT_LIST,
	SELECT_POSTRUN_REPORT_DETAILS,
	DELETE_CALIBRATION_HEAD,
	SELECT_CALIB_REPORT_BY_ID,
	SELECT_CALIB_REPORT_VALUES_BY_ID,
	SELECT_SYSTEM_SETTINGS_REPORT_LIST,
	SELECT_SYSTEM_SETTINGS_BY_ID,
	SELECT_METHOD_REPORT_SEARCH,
	SELECT_METHOD_REPORT_LIST,
	SELECT_RUN_REPORT_LIST,
	SELECT_RECIPE_HEADER_BY_ID,
	SELECT_RECIPE_VOLUME_BY_ID,
	SELECT_POSTRUN_RUN_BY_ID,
	SELECT_POSTRUN_METHOD_BY_RUN_ID,
	SELECT_POSTRUN_VOLUME_BY_METHOD_ID,
	SELECT_LINEAR_BY_ID,
	SELECT_LINEAR_REPORT_SEARCH,
	SELECT_LAST_LINEAR_REPORT,
	SELECT_LAST_POSTRUN_RUN,
	SELECT_LAST_PUMP_CALIBRATION,
	SELECT_SYSTEM_HISTORY_REPORT,
	SELECT_LINEAR_HISTORY_REPORT,
	SELECT_COMPLETE_METHOD_REPORT,
	SELECT_COMPLETE_METHOD_REPORT_VOLUMES,
	INSERT_USER,
	INSERT_USER_MGMT_HISTORY,
	ERROR_STATE
);
END_TYPE

// ---- POUs/MARCO/DB/STs/E_UserMgmtEventType.TcDUT
{attribute 'qualified_only'}
{attribute 'strict'}
TYPE E_UserMgmtEventType :
(
	None := 0,
    UserCreated := 1,
    UserDeleted := 2,
    GroupUpdated := 3,
    AutoLogoutUpdated := 4,
    UserUpdated := 5,
    PasswordChanged := 6
);
END_TYPE

// ---- POUs/MARCO/DB/STs/ST_CalibrationReportHeader.TcDUT
TYPE ST_CalibrationReportHeader :
STRUCT
	sReportId          : STRING(50);
    sCalibrationNo     : STRING(30);
    sUserId            : STRING(50);
    sDensity           : STRING(30);
    sSolventNo         : STRING(30);
    sSolventRevision   : STRING(30);
    sSysRevisionNo     : STRING(30);
    sAllowableFail     : STRING(30);
    sReplicates        : STRING(30);
    sCallInterval      : STRING(30);
    sCreatedAt         : STRING(30);
END_STRUCT
END_TYPE

// ---- POUs/MARCO/DB/STs/ST_CalibrationReportLine.TcDUT
TYPE ST_CalibrationReportLine :
STRUCT
	sDateTime           : STRING(40);
    sPumpNo             : STRING(10);
    sStep               : STRING(20);
    sTareWt             : STRING(30);
    sGrossWt            : STRING(30);
    sNetWt              : STRING(30);
    sNetVolume          : STRING(30);
    sTargetVolume       : STRING(30);
    sDifferencePercent  : STRING(30);
    sCriteria           : STRING(20);
    sPumpRevs           : STRING(30);
END_STRUCT
END_TYPE

// ---- POUs/MARCO/DB/STs/ST_CalibrationReportListItem.TcDUT
TYPE ST_CalibrationReportListItem :
STRUCT
	sReportId       : STRING(50);
    sCalibrationNo  : STRING(30);
    sCreatedAt      : STRING(30);
    sUserId         : STRING(50);
END_STRUCT
END_TYPE

// ---- POUs/MARCO/DB/STs/ST_Data_PCR.TcDUT
TYPE ST_Data_PCR :
STRUCT
	dateTime			: STRING(100);
	pumpNo				: STRING(100);
	step				: STRING(100);
	tareWt				: STRING(100);
	grossWt				: STRING(100);
	netVolume			: STRING(100);
	netWt				: STRING(100);
	targetVolume		: STRING(100);
	differencePercent	: STRING(100);
	criteria			: STRING(100);
	pumpRevs			: STRING(100);
	CalibrationNo		: INT;
	
END_STRUCT
END_TYPE

// ---- POUs/MARCO/DB/STs/ST_Data_UHR.TcDUT
TYPE ST_Data_UHR :
STRUCT
	userID				:STRING;
	accessLevel			:STRING;
	transactionType		:STRING;
	transactionDate		:STRING;
	transactedBy		:STRING;
END_STRUCT
END_TYPE

// ---- POUs/MARCO/DB/STs/ST_DB_Solvents.TcDUT
TYPE ST_DB_Solvents :
STRUCT
	solvent_ID   : DINT;

    solventName1 : STRING(80);
    density1     : STRING(40);

    addedBy      : STRING(80);
    addedDate    : STRING(40);

    solventName2 : STRING(80);
    solventName3 : STRING(80);
    solventName4 : STRING(80);

    density2     : STRING(40);
    density3     : STRING(40);
    density4     : STRING(40);
END_STRUCT
END_TYPE

// ---- POUs/MARCO/DB/STs/ST_LinearMotors.TcDUT
TYPE ST_LinearMotors :
STRUCT
	ID_Linear		: INT;
	pump1			: STRING(100);
	pump2			: STRING(100);
	pump3			: STRING(100);
	pump4			: STRING(100);
	pump5			: STRING(100);
	pump6			: STRING(100);
	pump7			: STRING(100);
	pump8			: STRING(100);
	pump9			: STRING(100);
	pump10			: STRING(100);
END_STRUCT
END_TYPE

// ---- POUs/MARCO/DB/STs/ST_ListMethod.TcDUT
TYPE ST_ListMethod :
STRUCT
	methodName		: STRING(100);
	methodRevision	: STRING(100);
	
END_STRUCT
END_TYPE

// ---- POUs/MARCO/DB/STs/ST_Parameters_MR.TcDUT
TYPE ST_Parameters_MR :
STRUCT
	methodName			: STRING(100);
	methodRevision		: STRING(100);
	methodCreatedBy		: STRING(100);
	methodCreatedOn		: STRING(100);
	solvent_R1			: STRING(100);
	solvent_R2			: STRING(100);
	solvent_W1			: STRING(100);
	solvent_W2			: STRING(100);
	time_R1				: STRING(100);
	time_R2				: STRING(100);
	time_W1				: STRING(100);
	time_W2				: STRING(100);	
	velocity_R1			: STRING(100);
	velocity_R2			: STRING(100);
	velocity_W1			: STRING(100);
	velocity_W2			: STRING(100);
	soakTime			: STRING(100);
	agitate_1_Time		: STRING(100);
	agitate_2_Time		: STRING(100);
	vialsToFill			: STRING(100);
	vialPrimeVol		: STRING(100);
	vial_1_FillVol		: STRING(100);
	vial_2_4_FillVol	: STRING(100);
	airDryTime			: STRING(100);
	methodID			: INT;
	methodStatus		: STRING(100);
	
END_STRUCT
END_TYPE

// ---- POUs/MARCO/DB/STs/ST_CompleteMethod.TcDUT
TYPE ST_CompleteMethod :
STRUCT
	methodName			: STRING(100);
	methodRevision		: STRING(100);
	methodCreatedBy		: STRING(100);
	methodCreatedOn		: STRING(100);
	solvent_R1			: STRING(100);
	solvent_R2			: STRING(100);
	solvent_W1			: STRING(100);
	solvent_W2			: STRING(100);
	time_R1				: STRING(100);
	time_R2				: STRING(100);
	time_W1				: STRING(100);
	time_W2				: STRING(100);	
	velocity_R1			: STRING(100);
	velocity_R2			: STRING(100);
	velocity_W1			: STRING(100);
	velocity_W2			: STRING(100);
	soakTime			: STRING(100);
	agitate_1_Time		: STRING(100);
	agitate_2_Time		: STRING(100);
	vialsToFill			: STRING(100);
	vialPrimeVol		: STRING(100);
	vial_1_FillVol		: STRING(100);
	vial_2_4_FillVol	: STRING(100);
	airDryTime			: STRING(100);
	methodID			: INT;
	methodStatus		: STRING(100);
	volumeData			: ARRAY[1..10] OF ST_VolumeData;
	
END_STRUCT
END_TYPE

// ---- POUs/MARCO/DB/STs/ST_Parameters_PCR.TcDUT
TYPE ST_Parameters_PCR :
STRUCT
	CalibrationNo		: INT;
    userID             	: STRING;
    density	            : STRING;
    solventNo           : STRING;
    solventRevision	    : STRING;
    allowableFail		: STRING;
    replicates	        : STRING;
    callInterval	    : STRING;
	sysRevisionNo		: INT;
END_STRUCT
END_TYPE

// ---- POUs/MARCO/DB/STs/ST_PostRunReport.TcDUT
TYPE ST_PostRunReport :
STRUCT
	runNo				: INT;
	analyst				: STRING(100);
	comment				: STRING(100);
	softwareVersion		: STRING(100);
	sysMasterRevision	: STRING(100);
	sysSettingsRevision	: STRING(100);
	meterVelocity		: STRING(100);
	runVelocity			: STRING(100);
	emptyTubesFactor	: STRING(100);
	fillTubesFactor		: STRING(100);
	solvent1NameRevision: STRING(100);
	solvent2NameRevision: STRING(100);
	solvent3NameRevision: STRING(100);
	solvent4NameRevision: STRING(100);
	timeEventStarted	: STRING(100);
	timeEventCompleted	: STRING(100);
	methodID			: INT;
	CalibrationNo		: INT;
END_STRUCT
END_TYPE

// ---- POUs/MARCO/DB/STs/ST_Solvents.TcDUT
TYPE ST_Solvents :
STRUCT
	Solvent_ID 		: INT;
	solventName1 	: STRING(100);
	solventName2 	: STRING(100);
	solventName3 	: STRING(100);
	solventName4 	: STRING(100);
	density1 		: STRING(100);
	density2 		: STRING(100);
	density3 		: STRING(100);
	density4 		: STRING(100);
	addedBy 		: STRING(100);
	addedDate 		: STRING(100);
END_STRUCT
END_TYPE

// ---- POUs/MARCO/DB/STs/ST_SysParameters.TcDUT
TYPE ST_SysParameters :
STRUCT
	gen_SealAndPump				: STRING(100);
	cal_AcceptanceCriteria		: STRING(100);
	cal_AllowableFail			: STRING(100);
	cal_Replicates				: STRING(100);
	cal_PumpCallIntervalDays	: STRING(100);
	cal_CloseAppOnCompletation	: STRING(100);
	AirDryTimeOnCompletation	: STRING(100);
	lkt_AllowableLeakTestFail	: STRING(100);
	lkt_LeakTestBuildupTime		: STRING(100);
	lkt_LeakTestHoldTime		: STRING(100);
	lkt_LeakTestPressure		: STRING(100);
	mec_PlatesClosedPosition	: STRING(100);
	mec_PlatesDryPosition		: STRING(100);
	mec_PlatesVelocity			: STRING(100);
	mec_MaxCurrentFastDown		: STRING(100);
	mec_MaxCurrentSlowDown		: STRING(100);
	mec_MaxCurrentSlowUp		: STRING(100);
	pmp_MeterVelocity			: STRING(100);
	pmp_RunVelocity				: STRING(100);
	pmp_EmptyFactor				: STRING(100);
	pmp_FillSolventTubesFactor	: STRING(100);
	smp_AboveCalibration		: STRING(100);
	smp_VialSetSpacing			: STRING(100);
	smp_IntoResBottom			: STRING(100);
	smp_IntoResDispense			: STRING(100);
	smp_IntoResWeigh			: STRING(100);
	smp_IntoVials				: STRING(100);
	sec_DisplayManualControl	: STRING(100);
	sec_CheckLogonEachRun		: STRING(100);
	createdBy					: STRING(100);
	createdDate					: STRING(100);
	sysRevisionNo				: INT;
	smp_AboveVialSet1			: STRING(100);
	smp_IntoWaste				: STRING(100);
	
END_STRUCT
END_TYPE

// ---- POUs/MARCO/DB/STs/ST_UserMgmtHistoryEvent.TcDUT
TYPE ST_UserMgmtHistoryEvent :
STRUCT
    bExecute            : BOOL;

    sTargetUser         : STRING(100);
    sEventType          : STRING(50);

    sOldGroup           : STRING(100);
    sNewGroup           : STRING(100);

    iOldAutoLogoutMin   : INT;
    iNewAutoLogoutMin   : INT;

    sPerformedBy        : STRING(100);
    sSourceScreen       : STRING(100);
    sEventComment       : STRING(255);

    bBusy               : BOOL;
    bDone               : BOOL;
    bError              : BOOL;
    sErrorText          : STRING(255);
END_STRUCT
END_TYPE

// ---- POUs/MARCO/DB/STs/ST_VolumeData.TcDUT
TYPE ST_VolumeData :
STRUCT
	VD_ID				: INT;
	pump				: STRING(100);
	stage				: STRING(100);
	rinse1				: STRING(100);
	rinse2				: STRING(100);
	wash1				: STRING(100);
	wash2				: STRING(100);
	methodID			: INT;
	
END_STRUCT
END_TYPE

// ---- GVLs/GVL_Alarms.TcGVL
{attribute 'qualified_only'}
VAR_GLOBAL

	arrEventText 	: ARRAY[0..400] OF T_MaxSTring;	// All events messages defined for the system - indices corresponds to indices of aEvents
	arrActiveEvents : ARRAY[0..400] OF T_MaxSTring;	// Active events messages - displayed in active alarms
	arrEventLogs	: ARRAY[0..400] OF T_MaxSTring;	// Logged events messages - displayed in alarm history
	arrEventFlag	: ARRAY[0..400] OF BOOL;		// Events triggers

